KUKA KRL program: EPS_2_251491_MH03A_A_20251118025156.src

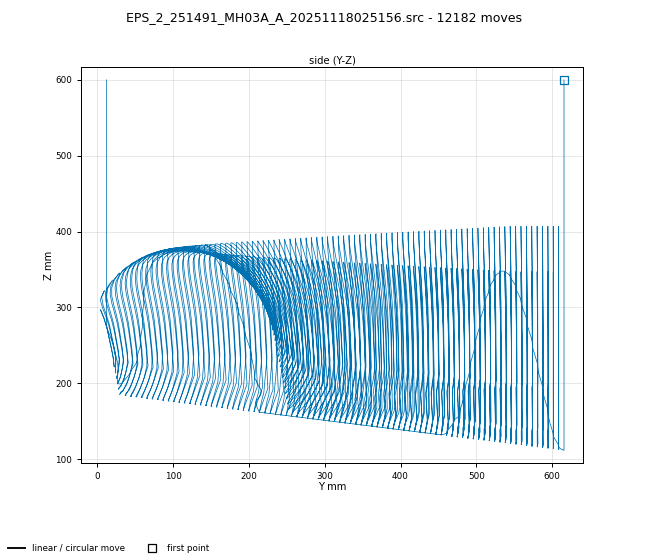
[picture p0: tool path of EPS_2_251491_MH03A_A_20251118025156.src, 12182 of 12184 moves have a stored position in this frame; points joined in program order, loops and branches not executed]
&ACCESS RVP
&REL 4
&COMMENT QRS 19112012
&PARAM EDITMASK = *
DEF PART()
EXT BAS (BAS_COMMAND :IN,REAL :IN )
INT I
BAS (#INITMOV,0 )

;KUKA QRS Post kuka4.cps  Date:22-06-2017 !

File_ID=2917

QRS_PRE_INIT()

;Init var - Until changes are made in qrs_pre_init
Outlet_Square_prg=0
Inlet_1_Square_prg=0
Inlet_2_Square_prg=0
Inlet_3_Square_prg=0
Inlet_4_Square_prg=0
Inlet_5_Square_prg=0

Outlet_1={X 0.000, Y 546.330, Z 306.500, B 0.000, E1 0.000 }
Inlet_1={X 0.000, Y 550.600, Z 246.500, B 0.000, E1 115.000 }
Outlet_1_type=201
Inlet_1_type=201
;QRS#1=Sidecore dimensions
;QRS#2=200-8" PVC SDR 35
;QRS#3=200-8" PVC SDR 35
;QRS#4=
;QRS#5=
;QRS#6=
;QRS#7=
;QRS#8=
;QRS#9=12-08 PSX
;QRS#10=12-08 PSX
;QRS#11=
;QRS#12=
;QRS#13=
;QRS#14=
;QRS#15=
;QRS#16=1220x127x686 2,25'
;QRS#17=EPS Height
;QRS#18=407
;QRS#19=*
;QRS#20= UPDATED VERSION 22-06-2017
;QRS#21=*
Outlet_Square=0100
Inlet_1_Square=0100
Inlet_2_Square=0
Inlet_3_Square=0
Inlet_4_Square=0
Inlet_5_Square=0
Mill_Square=1
Outlet_Square_Prg=204
Inlet_1_Square_prg=204

QRS_INIT()

$ADVANCE=5

; T1
PTP {E1 173.624,E2 173.624}
PTP {X 0,Y 615.49,A -85,B 0,C 180,E1 173.624,E2 173.624,E3 0,E4 0,E5 0,E6 0}
QRS_SPEED_INIT()
LIN {X 0,Y 615.49,Z 600,A -85,B 0,C 180,E1 173.624,E2 173.624,E3 0,E4 0,E5 0,E6 0} C_VEL
LIN {X 0,Y 615.49,Z 121.877,A -85,B 0,C 180,E1 173.624,E2 173.624} C_VEL
LIN {X 0,Y 615.49,Z 113.698,A -85,B 0,C 180,E1 173.624,E2 173.624} C_VEL
LIN {X 0,Y 615.469,Z 111.698,A -85,B 0,C 180,E1 173.438,E2 173.438} C_VEL
LIN {X 0,Y 615.485,Z 111.809,A -85,B 0,C 180,E1 172.29,E2 172.29} C_VEL
LIN {X 0,Y 615.448,Z 127.375,A -85,B 0,C 180,E1 169.473,E2 169.473} C_VEL
LIN {X 0,Y 615.475,Z 136.667,A -85,B 0,C 180,E1 167.805,E2 167.805} C_VEL
LIN {X 0,Y 615.485,Z 242.691,A -85,B 0,C 180,E1 166.547,E2 166.547} C_VEL
LIN {X 0,Y 615.49,Z 256.094,A -85,B 0,C 180,E1 166.252,E2 166.252} C_VEL
LIN {X 0,Y 615.493,Z 268.774,A -85,B 0,C 180,E1 165.836,E2 165.836} C_VEL
LIN {X 0,Y 615.466,Z 281.129,A -85,B 0,C 180,E1 165.282,E2 165.282} C_VEL
LIN {X 0,Y 615.476,Z 292.718,A -85,B 0,C 180,E1 164.604,E2 164.604} C_VEL
LIN {X 0,Y 615.498,Z 303.278,A -85,B 0,C 180,E1 163.831,E2 163.831} C_VEL
LIN {X 0,Y 615.498,Z 311.724,A -85,B 0,C 180,E1 163.072,E2 163.072} C_VEL
LIN {X 0,Y 615.498,Z 321.005,A -85,B 0,C 180,E1 162.044,E2 162.044} C_VEL
LIN {X 0,Y 615.496,Z 328.473,A -85,B 0,C 180,E1 161.009,E2 161.009} C_VEL
LIN {X 0,Y 615.497,Z 334.384,A -85,B 0,C 180,E1 159.968,E2 159.968} C_VEL
LIN {X 0,Y 615.495,Z 339.006,A -85,B 0,C 180,E1 158.92,E2 158.92} C_VEL
LIN {X 0,Y 615.492,Z 343.02,A -85,B 0,C 180,E1 157.653,E2 157.653} C_VEL
LIN {X 0,Y 615.496,Z 345.367,A -85,B 0,C 180,E1 156.444,E2 156.444} C_VEL
LIN {X 0,Y 615.493,Z 346.09,A -85,B 0,C 180,E1 155.729,E2 155.729} C_VEL
LIN {X 0,Y 615.498,Z 346.381,A -85,B 0,C 180,E1 155.009,E2 155.009} C_VEL
LIN {X 0,Y 615.496,Z 346.162,A -85,B 0,C 180,E1 154.285,E2 154.285} C_VEL
LIN {X 0,Y 615.497,Z 344.544,A -85,B 0,C 180,E1 152.954,E2 152.954} C_VEL
LIN {X 0,Y 615.492,Z 342.561,A -85,B 0,C 180,E1 152.085,E2 152.085} C_VEL
LIN {X 0,Y 615.496,Z 338.927,A -85,B 0,C 180,E1 150.969,E2 150.969} C_VEL
LIN {X 0,Y 615.497,Z 333.887,A -85,B 0,C 180,E1 149.841,E2 149.841} C_VEL
LIN {X 0,Y 615.494,Z 328.551,A -85,B 0,C 180,E1 148.913,E2 148.913} C_VEL
LIN {X 0,Y 615.495,Z 320.711,A -85,B 0,C 180,E1 147.83,E2 147.83} C_VEL
LIN {X 0,Y 615.498,Z 312.921,A -85,B 0,C 180,E1 146.96,E2 146.96} C_VEL
LIN {X 0,Y 615.497,Z 303.548,A -85,B 0,C 180,E1 146.101,E2 146.101} C_VEL
LIN {X 0,Y 615.487,Z 292.623,A -85,B 0,C 180,E1 145.3,E2 145.3} C_VEL
LIN {X 0,Y 615.492,Z 282.198,A -85,B 0,C 180,E1 144.686,E2 144.686} C_VEL
LIN {X 0,Y 615.486,Z 271.098,A -85,B 0,C 180,E1 144.167,E2 144.167} C_VEL
LIN {X 0,Y 615.458,Z 258.459,A -85,B 0,C 180,E1 143.722,E2 143.722} C_VEL
LIN {X 0,Y 615.456,Z 245.542,A -85,B 0,C 180,E1 143.415,E2 143.415} C_VEL
LIN {X 0,Y 615.467,Z 226.579,A -85,B 0,C 180,E1 143.161,E2 143.161} C_VEL
LIN {X 0,Y 615.448,Z 136.583,A -85,B 0,C 180,E1 142.089,E2 142.089} C_VEL
LIN {X 0,Y 615.481,Z 123.017,A -85,B 0,C 180,E1 139.654,E2 139.654} C_VEL
LIN {X 0,Y 615.467,Z 111.691,A -85,B 0,C 180,E1 137.559,E2 137.559} C_VEL
LIN {X 0,Y 615.495,Z 111.683,A -85,B 0,C 180,E1 134.933,E2 134.933} C_VEL
LIN {X 0,Y 615.482,Z 111.697,A -85,B 0,C 180,E1 132.08,E2 132.08} C_VEL
LIN {X 0,Y 615.466,Z 111.691,A -85,B 0,C 180,E1 129.752,E2 129.752} C_VEL
LIN {X 0,Y 615.488,Z 111.687,A -85,B 0,C 180,E1 126.937,E2 126.937} C_VEL
LIN {X 0,Y 615.47,Z 111.693,A -85,B 0,C 180,E1 124.023,E2 124.023} C_VEL
LIN {X 0,Y 615.469,Z 111.688,A -85,B 0,C 180,E1 121.687,E2 121.687} C_VEL
LIN {X 0,Y 615.486,Z 111.683,A -85,B 0,C 180,E1 119.407,E2 119.407} C_VEL
LIN {X 0,Y 615.481,Z 111.698,A -85,B 0,C 180,E1 116.445,E2 116.445} C_VEL
LIN {X 0,Y 615.485,Z 111.684,A -85,B 0,C 180,E1 113.557,E2 113.557} C_VEL
LIN {X 0,Y 615.48,Z 111.698,A -85,B 0,C 180,E1 110.556,E2 110.556} C_VEL
LIN {X 0,Y 615.473,Z 111.686,A -85,B 0,C 180,E1 107.958,E2 107.958} C_VEL
LIN {X 0,Y 615.486,Z 111.691,A -85,B 0,C 180,E1 105.226,E2 105.226} C_VEL
LIN {X 0,Y 615.471,Z 111.694,A -85,B 0,C 180,E1 102.531,E2 102.531} C_VEL
LIN {X 0,Y 615.492,Z 111.682,A -85,B 0,C 180,E1 99.862,E2 99.862} C_VEL
LIN {X 0,Y 615.49,Z 111.696,A -85,B 0,C 180,E1 97.216,E2 97.216} C_VEL
LIN {X 0,Y 615.469,Z 111.692,A -85,B 0,C 180,E1 94.585,E2 94.585} C_VEL
LIN {X 0,Y 615.499,Z 111.681,A -85,B 0,C 180,E1 91.963,E2 91.963} C_VEL
LIN {X 0,Y 615.491,Z 111.697,A -85,B 0,C 180,E1 89.346,E2 89.346} C_VEL
LIN {X 0,Y 615.469,Z 111.691,A -85,B 0,C 180,E1 86.727,E2 86.727} C_VEL
LIN {X 0,Y 615.498,Z 111.681,A -85,B 0,C 180,E1 84.102,E2 84.102} C_VEL
LIN {X 0,Y 615.494,Z 111.698,A -85,B 0,C 180,E1 81.464,E2 81.464} C_VEL
LIN {X 0,Y 615.469,Z 111.69,A -85,B 0,C 180,E1 78.807,E2 78.807} C_VEL
LIN {X 0,Y 615.487,Z 111.686,A -85,B 0,C 180,E1 76.066,E2 76.066} C_VEL
LIN {X 0,Y 615.483,Z 111.699,A -85,B 0,C 180,E1 73.414,E2 73.414} C_VEL
LIN {X 0,Y 615.481,Z 111.684,A -85,B 0,C 180,E1 70.662,E2 70.662} C_VEL
LIN {X 0,Y 615.487,Z 111.696,A -85,B 0,C 180,E1 67.864,E2 67.864} C_VEL
LIN {X 0,Y 615.471,Z 111.688,A -85,B 0,C 180,E1 65.008,E2 65.008} C_VEL
LIN {X 0,Y 615.479,Z 111.685,A -85,B 0,C 180,E1 62.823,E2 62.823} C_VEL
LIN {X 0,Y 615.499,Z 111.7,A -85,B 0,C 180,E1 59.841,E2 59.841} C_VEL
LIN {X 0,Y 615.475,Z 111.694,A -85,B 0,C 180,E1 57.542,E2 57.542} C_VEL
LIN {X 0,Y 615.471,Z 111.688,A -85,B 0,C 180,E1 55.184,E2 55.184} C_VEL
LIN {X 0,Y 615.493,Z 111.682,A -85,B 0,C 180,E1 52.759,E2 52.759} C_VEL
LIN {X 0,Y 615.487,Z 111.698,A -85,B 0,C 180,E1 49.911,E2 49.911} C_VEL
LIN {X 0,Y 615.47,Z 111.693,A -85,B 0,C 180,E1 47.646,E2 47.646} C_VEL
LIN {X 0,Y 615.495,Z 111.682,A -85,B 0,C 180,E1 44.933,E2 44.933} C_VEL
LIN {X 0,Y 615.488,Z 111.698,A -85,B 0,C 180,E1 42.081,E2 42.081} C_VEL
LIN {X 0,Y 615.469,Z 111.691,A -85,B 0,C 180,E1 39.751,E2 39.751} C_VEL
LIN {X 0,Y 615.487,Z 111.686,A -85,B 0,C 180,E1 36.937,E2 36.937} C_VEL
LIN {X 0,Y 615.474,Z 111.694,A -85,B 0,C 180,E1 34.022,E2 34.022} C_VEL
LIN {X 0,Y 615.471,Z 111.688,A -85,B 0,C 180,E1 31.686,E2 31.686} C_VEL
LIN {X 0,Y 615.487,Z 111.683,A -85,B 0,C 180,E1 29.406,E2 29.406} C_VEL
LIN {X 0,Y 615.485,Z 111.699,A -85,B 0,C 180,E1 26.444,E2 26.444} C_VEL
LIN {X 0,Y 615.485,Z 111.683,A -85,B 0,C 180,E1 23.556,E2 23.556} C_VEL
LIN {X 0,Y 615.483,Z 111.699,A -85,B 0,C 180,E1 20.557,E2 20.557} C_VEL
LIN {X 0,Y 615.475,Z 111.686,A -85,B 0,C 180,E1 17.957,E2 17.957} C_VEL
LIN {X 0,Y 615.482,Z 111.691,A -85,B 0,C 180,E1 15.226,E2 15.226} C_VEL
LIN {X 0,Y 615.477,Z 111.694,A -85,B 0,C 180,E1 12.53,E2 12.53} C_VEL
LIN {X 0,Y 615.493,Z 111.681,A -85,B 0,C 180,E1 9.862,E2 9.862} C_VEL
LIN {X 0,Y 615.486,Z 111.695,A -85,B 0,C 180,E1 7.215,E2 7.215} C_VEL
LIN {X 0,Y 615.473,Z 111.692,A -85,B 0,C 180,E1 4.584,E2 4.584} C_VEL
LIN {X 0,Y 615.5,Z 111.68,A -85,B 0,C 180,E1 1.963,E2 1.963} C_VEL
LIN {X 0,Y 615.488,Z 111.695,A -85,B 0,C 180,E1 -0.654,E2 -0.654} C_VEL
LIN {X 0,Y 615.473,Z 111.692,A -85,B 0,C 180,E1 -3.273,E2 -3.273} C_VEL
LIN {X 0,Y 615.498,Z 111.681,A -85,B 0,C 180,E1 -5.899,E2 -5.899} C_VEL
LIN {X 0,Y 615.49,Z 111.697,A -85,B 0,C 180,E1 -8.537,E2 -8.537} C_VEL
LIN {X 0,Y 615.472,Z 111.69,A -85,B 0,C 180,E1 -11.194,E2 -11.194} C_VEL
LIN {X 0,Y 615.486,Z 111.686,A -85,B 0,C 180,E1 -13.933,E2 -13.933} C_VEL
LIN {X 0,Y 615.486,Z 111.701,A -85,B 0,C 180,E1 -16.587,E2 -16.587} C_VEL
LIN {X 0,Y 615.482,Z 111.684,A -85,B 0,C 180,E1 -19.338,E2 -19.338} C_VEL
LIN {X 0,Y 615.483,Z 111.695,A -85,B 0,C 180,E1 -22.137,E2 -22.137} C_VEL
LIN {X 0,Y 615.474,Z 111.688,A -85,B 0,C 180,E1 -24.993,E2 -24.993} C_VEL
LIN {X 0,Y 615.481,Z 111.684,A -85,B 0,C 180,E1 -27.178,E2 -27.178} C_VEL
LIN {X 0,Y 615.482,Z 111.69,A -85,B 0,C 180,E1 -29.794,E2 -29.794} C_VEL
LIN {X 0,Y 615.479,Z 111.695,A -85,B 0,C 180,E1 -32.458,E2 -32.458} C_VEL
LIN {X 0,Y 615.475,Z 111.687,A -85,B 0,C 180,E1 -34.816,E2 -34.816} C_VEL
LIN {X 0,Y 615.493,Z 111.682,A -85,B 0,C 180,E1 -37.242,E2 -37.242} C_VEL
LIN {X 0,Y 615.493,Z 111.699,A -85,B 0,C 180,E1 -40.09,E2 -40.09} C_VEL
LIN {X 0,Y 615.488,Z 111.683,A -85,B 0,C 180,E1 -43.048,E2 -43.048} C_VEL
LIN {X 0,Y 615.49,Z 111.698,A -85,B 0,C 180,E1 -46.003,E2 -46.003} C_VEL
LIN {X 0,Y 615.487,Z 111.683,A -85,B 0,C 180,E1 -48.906,E2 -48.906} C_VEL
LIN {X 0,Y 615.485,Z 111.697,A -85,B 0,C 180,E1 -51.932,E2 -51.932} C_VEL
LIN {X 0,Y 615.472,Z 111.688,A -85,B 0,C 180,E1 -54.383,E2 -54.383} C_VEL
LIN {X 0,Y 615.487,Z 111.683,A -85,B 0,C 180,E1 -56.764,E2 -56.764} C_VEL
LIN {X 0,Y 615.482,Z 111.689,A -85,B 0,C 180,E1 -59.08,E2 -59.08} C_VEL
LIN {X 0,Y 615.496,Z 111.701,A -85,B 0,C 180,E1 -61.549,E2 -61.549} C_VEL
LIN {X 0,Y 615.485,Z 111.683,A -85,B 0,C 180,E1 -64.432,E2 -64.432} C_VEL
LIN {X 0,Y 615.488,Z 111.875,A -85,B 0,C 180,E1 -66.711,E2 -66.711} C_VEL
LIN {X 0,Y 615.45,Z 133.105,A -85,B 0,C 180,E1 -69.453,E2 -69.453} C_VEL
LIN {X 0,Y 615.494,Z 154.838,A -85,B 0,C 180,E1 -72.215,E2 -72.215} C_VEL
LIN {X 0,Y 615.485,Z 176.626,A -85,B 0,C 180,E1 -74.944,E2 -74.944} C_VEL
LIN {X 0,Y 615.449,Z 194.138,A -85,B 0,C 180,E1 -77.113,E2 -77.113} C_VEL
LIN {X 0,Y 615.488,Z 302.845,A -85,B 0,C 180,E1 -78.411,E2 -78.411} C_VEL
LIN {X 0,Y 615.477,Z 315.355,A -85,B 0,C 180,E1 -78.682,E2 -78.682} C_VEL
LIN {X 0,Y 615.488,Z 328.618,A -85,B 0,C 180,E1 -79.113,E2 -79.113} C_VEL
LIN {X 0,Y 615.477,Z 340.484,A -85,B 0,C 180,E1 -79.639,E2 -79.639} C_VEL
LIN {X 0,Y 615.494,Z 351.998,A -85,B 0,C 180,E1 -80.304,E2 -80.304} C_VEL
LIN {X 0,Y 615.499,Z 362.344,A -85,B 0,C 180,E1 -81.05,E2 -81.05} C_VEL
LIN {X 0,Y 615.497,Z 370.814,A -85,B 0,C 180,E1 -81.794,E2 -81.794} C_VEL
LIN {X 0,Y 615.498,Z 378.608,A -85,B 0,C 180,E1 -82.62,E2 -82.62} C_VEL
LIN {X 0,Y 615.496,Z 386.205,A -85,B 0,C 180,E1 -83.608,E2 -83.608} C_VEL
LIN {X 0,Y 615.498,Z 393.206,A -85,B 0,C 180,E1 -84.759,E2 -84.759} C_VEL
LIN {X 0,Y 615.494,Z 397.852,A -85,B 0,C 180,E1 -85.744,E2 -85.744} C_VEL
LIN {X 0,Y 615.494,Z 401.399,A -85,B 0,C 180,E1 -86.727,E2 -86.727} C_VEL
LIN {X 0,Y 615.497,Z 403.234,A -85,B 0,C 180,E1 -87.382,E2 -87.382} C_VEL
LIN {X 0,Y 615.5,Z 404.608,A -85,B 0,C 180,E1 -88.037,E2 -88.037} C_VEL
LIN {X 0,Y 615.496,Z 406.174,A -85,B 0,C 180,E1 -89.346,E2 -89.346} C_VEL
LIN {X 0,Y 615.494,Z 406.389,A -85,B 0,C 180,E1 -90,E2 -90} C_VEL
LIN {X 0,Y 615.495,Z 405.58,A -85,B 0,C 180,E1 -91.309,E2 -91.309} C_VEL
LIN {X 0,Y 615.5,Z 404.607,A -85,B 0,C 180,E1 -91.963,E2 -91.963} C_VEL
LIN {X 0,Y 615.497,Z 403.232,A -85,B 0,C 180,E1 -92.618,E2 -92.618} C_VEL
LIN {X 0,Y 615.496,Z 400.349,A -85,B 0,C 180,E1 -93.601,E2 -93.601} C_VEL
LIN {X 0,Y 615.498,Z 396.44,A -85,B 0,C 180,E1 -94.585,E2 -94.585} C_VEL
LIN {X 0,Y 615.499,Z 391.404,A -85,B 0,C 180,E1 -95.57,E2 -95.57} C_VEL
LIN {X 0,Y 615.497,Z 384.87,A -85,B 0,C 180,E1 -96.583,E2 -96.583} C_VEL
LIN {X 0,Y 615.497,Z 377.131,A -85,B 0,C 180,E1 -97.546,E2 -97.546} C_VEL
LIN {X 0,Y 615.498,Z 369.042,A -85,B 0,C 180,E1 -98.371,E2 -98.371} C_VEL
LIN {X 0,Y 615.499,Z 359.164,A -85,B 0,C 180,E1 -99.199,E2 -99.199} C_VEL
LIN {X 0,Y 615.488,Z 347.977,A -85,B 0,C 180,E1 -99.945,E2 -99.945} C_VEL
LIN {X 0,Y 615.482,Z 337.018,A -85,B 0,C 180,E1 -100.527,E2 -100.527} C_VEL
LIN {X 0,Y 615.48,Z 324.487,A -85,B 0,C 180,E1 -101.04,E2 -101.04} C_VEL
LIN {X 0,Y 615.479,Z 312.057,A -85,B 0,C 180,E1 -101.402,E2 -101.402} C_VEL
LIN {X 0,Y 615.493,Z 298.448,A -85,B 0,C 180,E1 -101.652,E2 -101.652} C_VEL
LIN {X 0,Y 615.449,Z 194.134,A -85,B 0,C 180,E1 -102.887,E2 -102.887} C_VEL
LIN {X 0,Y 615.493,Z 171.173,A -85,B 0,C 180,E1 -105.735,E2 -105.735} C_VEL
LIN {X 0,Y 615.469,Z 149.687,A -85,B 0,C 180,E1 -108.436,E2 -108.436} C_VEL
LIN {X 0,Y 615.496,Z 127.565,A -85,B 0,C 180,E1 -111.256,E2 -111.256} C_VEL
LIN {X 0,Y 615.49,Z 111.683,A -85,B 0,C 180,E1 -113.334,E2 -113.334} C_VEL
LIN {X 0,Y 615.481,Z 111.686,A -85,B 0,C 180,E1 -115.716,E2 -115.716} C_VEL
LIN {X 0,Y 615.496,Z 111.699,A -85,B 0,C 180,E1 -118.451,E2 -118.451} C_VEL
LIN {X 0,Y 615.485,Z 111.685,A -85,B 0,C 180,E1 -121.085,E2 -121.085} C_VEL
LIN {X 0,Y 615.483,Z 111.686,A -85,B 0,C 180,E1 -123.533,E2 -123.533} C_VEL
LIN {X 0,Y 615.48,Z 111.695,A -85,B 0,C 180,E1 -126.425,E2 -126.425} C_VEL
LIN {X 0,Y 615.494,Z 111.681,A -85,B 0,C 180,E1 -129.062,E2 -129.062} C_VEL
LIN {X 0,Y 615.488,Z 111.699,A -85,B 0,C 180,E1 -132.08,E2 -132.08} C_VEL
LIN {X 0,Y 615.495,Z 111.682,A -85,B 0,C 180,E1 -135.068,E2 -135.068} C_VEL
LIN {X 0,Y 615.489,Z 111.698,A -85,B 0,C 180,E1 -137.92,E2 -137.92} C_VEL
LIN {X 0,Y 615.469,Z 111.692,A -85,B 0,C 180,E1 -140.248,E2 -140.248} C_VEL
LIN {X 0,Y 615.488,Z 111.687,A -85,B 0,C 180,E1 -143.064,E2 -143.064} C_VEL
LIN {X 0,Y 615.47,Z 111.693,A -85,B 0,C 180,E1 -145.977,E2 -145.977} C_VEL
LIN {X 0,Y 615.468,Z 111.688,A -85,B 0,C 180,E1 -148.313,E2 -148.313} C_VEL
LIN {X 0,Y 615.486,Z 111.684,A -85,B 0,C 180,E1 -150.593,E2 -150.593} C_VEL
LIN {X 0,Y 615.477,Z 111.697,A -85,B 0,C 180,E1 -153.555,E2 -153.555} C_VEL
LIN {X 0,Y 615.464,Z 111.689,A -85,B 0,C 180,E1 -155.997,E2 -155.997} C_VEL
LIN {X 0,Y 615.495,Z 111.685,A -85,B 0,C 180,E1 -158.568,E2 -158.568} C_VEL
LIN {X 0,Y 615.47,Z 111.696,A -85,B 0,C 180,E1 -161.401,E2 -161.401} C_VEL
LIN {X 0,Y 615.475,Z 111.686,A -85,B 0,C 180,E1 -164.094,E2 -164.094} C_VEL
LIN {X 0,Y 615.493,Z 111.698,A -85,B 0,C 180,E1 -166.799,E2 -166.799} C_VEL
LIN {X 0,Y 615.455,Z 111.693,A -85,B 0,C 180,E1 -169.472,E2 -169.472} C_VEL
LIN {X 0,Y 615.484,Z 111.687,A -85,B 0,C 180,E1 -172.124,E2 -172.124} C_VEL
LIN {X 0,Y 615.488,Z 111.699,A -85,B 0,C 180,E1 -174.759,E2 -174.759} C_VEL
LIN {X 0,Y 615.452,Z 111.692,A -85,B 0,C 180,E1 -177.382,E2 -177.382} C_VEL
LIN {X 0,Y 615.487,Z 111.688,A -85,B 0,C 180,E1 -180,E2 -180} C_VEL
LIN {X 0,Y 615.477,Z 111.698,A -85,B 0,C 180,E1 -182.618,E2 -182.618} C_VEL
LIN {X 0,Y 615.447,Z 111.692,A -85,B 0,C 180,E1 -185.241,E2 -185.241} C_VEL
LIN {X 0,Y 615.469,Z 111.698,A -85,B 0,C 180,E1 -186.562,E2 -186.562} C_VEL
LIN {X 0,Y 614.782,Z 111.892,A -85,B 0,C 180,E1 -186.929,E2 -186.929} C_VEL
LIN {X 0,Y 611.98,Z 112.983,A -85,B 0,C 180,E1 -187.496,E2 -187.496} C_VEL
LIN {X 0,Y 609.163,Z 115.021,A -85,B 0,C 180,E1 -188.047,E2 -188.047} C_VEL
LIN {X 0,Y 608.467,Z 116.714,A -85,B 0,C 180,E1 -188.385,E2 -188.385} C_VEL
LIN {X 0,Y 608.47,Z 131.376,A -85,B 0,C 180,E1 -191.052,E2 -191.052} C_VEL
LIN {X 0,Y 608.452,Z 136.863,A -85,B 0,C 180,E1 -192.042,E2 -192.042} C_VEL
LIN {X 0,Y 608.548,Z 243.573,A -85,B 0,C 180,E1 -193.333,E2 -193.333} C_VEL
LIN {X 0,Y 608.539,Z 256.703,A -85,B 0,C 180,E1 -193.631,E2 -193.631} C_VEL
LIN {X 0,Y 608.522,Z 268.854,A -85,B 0,C 180,E1 -194.036,E2 -194.036} C_VEL
LIN {X 0,Y 608.487,Z 280.346,A -85,B 0,C 180,E1 -194.549,E2 -194.549} C_VEL
LIN {X 0,Y 608.457,Z 292.172,A -85,B 0,C 180,E1 -195.234,E2 -195.234} C_VEL
LIN {X 0,Y 608.477,Z 302.792,A -85,B 0,C 180,E1 -196.007,E2 -196.007} C_VEL
LIN {X 0,Y 608.461,Z 311.53,A -85,B 0,C 180,E1 -196.784,E2 -196.784} C_VEL
LIN {X 0,Y 608.458,Z 320.967,A -85,B 0,C 180,E1 -197.823,E2 -197.823} C_VEL
LIN {X 0,Y 608.447,Z 328.574,A -85,B 0,C 180,E1 -198.87,E2 -198.87} C_VEL
LIN {X 0,Y 608.436,Z 334.624,A -85,B 0,C 180,E1 -199.922,E2 -199.922} C_VEL
LIN {X 0,Y 608.426,Z 339.347,A -85,B 0,C 180,E1 -200.982,E2 -200.982} C_VEL
LIN {X 0,Y 608.454,Z 342.881,A -85,B 0,C 180,E1 -202.048,E2 -202.048} C_VEL
LIN {X 0,Y 608.423,Z 345.311,A -85,B 0,C 180,E1 -203.125,E2 -203.125} C_VEL
LIN {X 0,Y 608.42,Z 346.613,A -85,B 0,C 180,E1 -204.14,E2 -204.14} C_VEL
LIN {X 0,Y 608.439,Z 346.946,A -85,B 0,C 180,E1 -205.301,E2 -205.301} C_VEL
LIN {X 0,Y 608.425,Z 346.552,A -85,B 0,C 180,E1 -206.036,E2 -206.036} C_VEL
LIN {X 0,Y 608.437,Z 344.89,A -85,B 0,C 180,E1 -207.199,E2 -207.199} C_VEL
LIN {X 0,Y 608.427,Z 341.138,A -85,B 0,C 180,E1 -208.612,E2 -208.612} C_VEL
LIN {X 0,Y 608.446,Z 336.505,A -85,B 0,C 180,E1 -209.78,E2 -209.78} C_VEL
LIN {X 0,Y 608.454,Z 330.52,A -85,B 0,C 180,E1 -210.904,E2 -210.904} C_VEL
LIN {X 0,Y 608.466,Z 323.827,A -85,B 0,C 180,E1 -211.899,E2 -211.899} C_VEL
LIN {X 0,Y 608.479,Z 315.688,A -85,B 0,C 180,E1 -212.878,E2 -212.878} C_VEL
LIN {X 0,Y 608.489,Z 306.888,A -85,B 0,C 180,E1 -213.737,E2 -213.737} C_VEL
LIN {X 0,Y 608.477,Z 296.262,A -85,B 0,C 180,E1 -214.578,E2 -214.578} C_VEL
LIN {X 0,Y 608.494,Z 285.309,A -85,B 0,C 180,E1 -215.274,E2 -215.274} C_VEL
LIN {X 0,Y 608.515,Z 273,A -85,B 0,C 180,E1 -215.883,E2 -215.883} C_VEL
LIN {X 0,Y 608.502,Z 260.618,A -85,B 0,C 180,E1 -216.344,E2 -216.344} C_VEL
LIN {X 0,Y 608.501,Z 247.794,A -85,B 0,C 180,E1 -216.679,E2 -216.679} C_VEL
LIN {X 0,Y 608.53,Z 232.344,A -85,B 0,C 180,E1 -216.909,E2 -216.909} C_VEL
LIN {X 0,Y 608.416,Z 136.878,A -85,B 0,C 180,E1 -218.046,E2 -218.046} C_VEL
LIN {X 0,Y 608.482,Z 123.216,A -85,B 0,C 180,E1 -220.517,E2 -220.517} C_VEL
LIN {X 0,Y 608.449,Z 112.69,A -85,B 0,C 180,E1 -222.445,E2 -222.445} C_VEL
LIN {X 0,Y 608.462,Z 112.688,A -85,B 0,C 180,E1 -225.204,E2 -225.204} C_VEL
LIN {X 0,Y 608.462,Z 112.693,A -85,B 0,C 180,E1 -227.938,E2 -227.938} C_VEL
LIN {X 0,Y 608.448,Z 112.688,A -85,B 0,C 180,E1 -230.705,E2 -230.705} C_VEL
LIN {X 0,Y 608.459,Z 112.689,A -85,B 0,C 180,E1 -233.085,E2 -233.085} C_VEL
LIN {X 0,Y 608.466,Z 112.696,A -85,B 0,C 180,E1 -235.53,E2 -235.53} C_VEL
LIN {X 0,Y 608.461,Z 112.69,A -85,B 0,C 180,E1 -237.905,E2 -237.905} C_VEL
LIN {X 0,Y 608.455,Z 112.688,A -85,B 0,C 180,E1 -240.22,E2 -240.22} C_VEL
LIN {X 0,Y 608.48,Z 112.686,A -85,B 0,C 180,E1 -242.792,E2 -242.792} C_VEL
LIN {X 0,Y 608.447,Z 112.697,A -85,B 0,C 180,E1 -245.428,E2 -245.428} C_VEL
LIN {X 0,Y 608.467,Z 112.686,A -85,B 0,C 180,E1 -248.308,E2 -248.308} C_VEL
LIN {X 0,Y 608.468,Z 112.695,A -85,B 0,C 180,E1 -251.284,E2 -251.284} C_VEL
LIN {X 0,Y 608.451,Z 112.688,A -85,B 0,C 180,E1 -253.906,E2 -253.906} C_VEL
LIN {X 0,Y 608.464,Z 112.689,A -85,B 0,C 180,E1 -256.643,E2 -256.643} C_VEL
LIN {X 0,Y 608.455,Z 112.692,A -85,B 0,C 180,E1 -259.35,E2 -259.35} C_VEL
LIN {X 0,Y 608.475,Z 112.685,A -85,B 0,C 180,E1 -262.033,E2 -262.033} C_VEL
LIN {X 0,Y 608.468,Z 112.692,A -85,B 0,C 180,E1 -264.698,E2 -264.698} C_VEL
LIN {X 0,Y 608.463,Z 112.689,A -85,B 0,C 180,E1 -267.352,E2 -267.352} C_VEL
LIN {X 0,Y 608.477,Z 112.685,A -85,B 0,C 180,E1 -270,E2 -270} C_VEL
LIN {X 0,Y 608.478,Z 112.693,A -85,B 0,C 180,E1 -272.648,E2 -272.648} C_VEL
LIN {X 0,Y 608.451,Z 112.689,A -85,B 0,C 180,E1 -275.302,E2 -275.302} C_VEL
LIN {X 0,Y 608.479,Z 112.685,A -85,B 0,C 180,E1 -277.967,E2 -277.967} C_VEL
LIN {X 0,Y 608.463,Z 112.69,A -85,B 0,C 180,E1 -280.954,E2 -280.954} C_VEL
LIN {X 0,Y 608.453,Z 112.688,A -85,B 0,C 180,E1 -283.356,E2 -283.356} C_VEL
LIN {X 0,Y 608.462,Z 112.691,A -85,B 0,C 180,E1 -286.093,E2 -286.093} C_VEL
LIN {X 0,Y 608.452,Z 112.691,A -85,B 0,C 180,E1 -288.869,E2 -288.869} C_VEL
LIN {X 0,Y 608.472,Z 112.686,A -85,B 0,C 180,E1 -291.691,E2 -291.691} C_VEL
LIN {X 0,Y 608.448,Z 112.694,A -85,B 0,C 180,E1 -294.571,E2 -294.571} C_VEL
LIN {X 0,Y 608.472,Z 112.685,A -85,B 0,C 180,E1 -297.207,E2 -297.207} C_VEL
LIN {X 0,Y 608.47,Z 112.692,A -85,B 0,C 180,E1 -299.972,E2 -299.972} C_VEL
LIN {X 0,Y 608.452,Z 112.691,A -85,B 0,C 180,E1 -302.521,E2 -302.521} C_VEL
LIN {X 0,Y 608.438,Z 112.689,A -85,B 0,C 180,E1 -304.904,E2 -304.904} C_VEL
LIN {X 0,Y 608.479,Z 112.684,A -85,B 0,C 180,E1 -307.16,E2 -307.16} C_VEL
LIN {X 0,Y 608.476,Z 112.687,A -85,B 0,C 180,E1 -309.439,E2 -309.439} C_VEL
LIN {X 0,Y 608.442,Z 112.692,A -85,B 0,C 180,E1 -312.333,E2 -312.333} C_VEL
LIN {X 0,Y 608.459,Z 112.687,A -85,B 0,C 180,E1 -314.795,E2 -314.795} C_VEL
LIN {X 0,Y 608.462,Z 112.695,A -85,B 0,C 180,E1 -317.665,E2 -317.665} C_VEL
LIN {X 0,Y 608.475,Z 112.685,A -85,B 0,C 180,E1 -320.701,E2 -320.701} C_VEL
LIN {X 0,Y 608.458,Z 112.689,A -85,B 0,C 180,E1 -323.086,E2 -323.086} C_VEL
LIN {X 0,Y 608.466,Z 112.695,A -85,B 0,C 180,E1 -325.531,E2 -325.531} C_VEL
LIN {X 0,Y 608.465,Z 112.691,A -85,B 0,C 180,E1 -327.906,E2 -327.906} C_VEL
LIN {X 0,Y 608.455,Z 112.688,A -85,B 0,C 180,E1 -330.22,E2 -330.22} C_VEL
LIN {X 0,Y 608.478,Z 112.685,A -85,B 0,C 180,E1 -332.792,E2 -332.792} C_VEL
LIN {X 0,Y 608.447,Z 112.699,A -85,B 0,C 180,E1 -335.429,E2 -335.429} C_VEL
LIN {X 0,Y 608.468,Z 112.686,A -85,B 0,C 180,E1 -338.309,E2 -338.309} C_VEL
LIN {X 0,Y 608.469,Z 112.696,A -85,B 0,C 180,E1 -341.283,E2 -341.283} C_VEL
LIN {X 0,Y 608.453,Z 112.688,A -85,B 0,C 180,E1 -343.906,E2 -343.906} C_VEL
LIN {X 0,Y 608.462,Z 112.689,A -85,B 0,C 180,E1 -346.644,E2 -346.644} C_VEL
LIN {X 0,Y 608.458,Z 112.693,A -85,B 0,C 180,E1 -349.35,E2 -349.35} C_VEL
LIN {X 0,Y 608.476,Z 112.685,A -85,B 0,C 180,E1 -352.033,E2 -352.033} C_VEL
LIN {X 0,Y 608.464,Z 112.692,A -85,B 0,C 180,E1 -354.698,E2 -354.698} C_VEL
LIN {X 0,Y 608.466,Z 112.69,A -85,B 0,C 180,E1 -357.352,E2 -357.352} C_VEL
LIN {X 0,Y 608.477,Z 112.685,A -85,B 0,C 180,E1 -360,E2 -360} C_VEL
LIN {X 0,Y 608.473,Z 112.692,A -85,B 0,C 180,E1 -362.648,E2 -362.648} C_VEL
LIN {X 0,Y 608.454,Z 112.69,A -85,B 0,C 180,E1 -365.302,E2 -365.302} C_VEL
LIN {X 0,Y 608.479,Z 112.685,A -85,B 0,C 180,E1 -367.967,E2 -367.967} C_VEL
LIN {X 0,Y 608.466,Z 112.691,A -85,B 0,C 180,E1 -370.956,E2 -370.956} C_VEL
LIN {X 0,Y 608.455,Z 112.688,A -85,B 0,C 180,E1 -373.357,E2 -373.357} C_VEL
LIN {X 0,Y 608.461,Z 112.69,A -85,B 0,C 180,E1 -376.094,E2 -376.094} C_VEL
LIN {X 0,Y 608.455,Z 112.691,A -85,B 0,C 180,E1 -378.87,E2 -378.87} C_VEL
LIN {X 0,Y 608.471,Z 112.686,A -85,B 0,C 180,E1 -381.692,E2 -381.692} C_VEL
LIN {X 0,Y 608.45,Z 112.694,A -85,B 0,C 180,E1 -384.571,E2 -384.571} C_VEL
LIN {X 0,Y 608.474,Z 112.685,A -85,B 0,C 180,E1 -387.207,E2 -387.207} C_VEL
LIN {X 0,Y 608.468,Z 112.692,A -85,B 0,C 180,E1 -389.972,E2 -389.972} C_VEL
LIN {X 0,Y 608.455,Z 112.688,A -85,B 0,C 180,E1 -392.88,E2 -392.88} C_VEL
LIN {X 0,Y 608.435,Z 112.69,A -85,B 0,C 180,E1 -395.278,E2 -395.278} C_VEL
LIN {X 0,Y 608.471,Z 112.69,A -85,B 0,C 180,E1 -397.746,E2 -397.746} C_VEL
LIN {X 0,Y 608.449,Z 112.693,A -85,B 0,C 180,E1 -400.329,E2 -400.329} C_VEL
LIN {X 0,Y 608.453,Z 112.687,A -85,B 0,C 180,E1 -402.96,E2 -402.96} C_VEL
LIN {X 0,Y 608.465,Z 112.694,A -85,B 0,C 180,E1 -405.736,E2 -405.736} C_VEL
LIN {X 0,Y 608.457,Z 112.687,A -85,B 0,C 180,E1 -408.659,E2 -408.659} C_VEL
LIN {X 0,Y 608.469,Z 112.69,A -85,B 0,C 180,E1 -411.412,E2 -411.412} C_VEL
LIN {X 0,Y 608.445,Z 112.695,A -85,B 0,C 180,E1 -413.955,E2 -413.955} C_VEL
LIN {X 0,Y 608.447,Z 112.689,A -85,B 0,C 180,E1 -416.329,E2 -416.329} C_VEL
LIN {X 0,Y 608.448,Z 112.688,A -85,B 0,C 180,E1 -418.733,E2 -418.733} C_VEL
LIN {X 0,Y 608.476,Z 112.692,A -85,B 0,C 180,E1 -421.38,E2 -421.38} C_VEL
LIN {X 0,Y 608.443,Z 112.692,A -85,B 0,C 180,E1 -423.965,E2 -423.965} C_VEL
LIN {X 0,Y 608.467,Z 112.728,A -85,B 0,C 180,E1 -426.539,E2 -426.539} C_VEL
LIN {X 0,Y 608.595,Z 127.57,A -85,B 0,C 180,E1 -428.491,E2 -428.491} C_VEL
LIN {X 0,Y 608.498,Z 149.174,A -85,B 0,C 180,E1 -431.277,E2 -431.277} C_VEL
LIN {X 0,Y 608.495,Z 168.58,A -85,B 0,C 180,E1 -433.744,E2 -433.744} C_VEL
LIN {X 0,Y 608.479,Z 190.348,A -85,B 0,C 180,E1 -436.474,E2 -436.474} C_VEL
LIN {X 0,Y 608.446,Z 194.357,A -85,B 0,C 180,E1 -436.973,E2 -436.973} C_VEL
LIN {X 0,Y 608.546,Z 302.961,A -85,B 0,C 180,E1 -438.277,E2 -438.277} C_VEL
LIN {X 0,Y 608.512,Z 316.226,A -85,B 0,C 180,E1 -438.572,E2 -438.572} C_VEL
LIN {X 0,Y 608.514,Z 328.631,A -85,B 0,C 180,E1 -438.982,E2 -438.982} C_VEL
LIN {X 0,Y 608.499,Z 340.64,A -85,B 0,C 180,E1 -439.519,E2 -439.519} C_VEL
LIN {X 0,Y 608.484,Z 352.201,A -85,B 0,C 180,E1 -440.191,E2 -440.191} C_VEL
LIN {X 0,Y 608.485,Z 362.597,A -85,B 0,C 180,E1 -440.946,E2 -440.946} C_VEL
LIN {X 0,Y 608.475,Z 371.114,A -85,B 0,C 180,E1 -441.699,E2 -441.699} C_VEL
LIN {X 0,Y 608.471,Z 378.962,A -85,B 0,C 180,E1 -442.534,E2 -442.534} C_VEL
LIN {X 0,Y 608.46,Z 386.288,A -85,B 0,C 180,E1 -443.485,E2 -443.485} C_VEL
LIN {X 0,Y 608.451,Z 391.867,A -85,B 0,C 180,E1 -444.366,E2 -444.366} C_VEL
LIN {X 0,Y 608.432,Z 396.951,A -85,B 0,C 180,E1 -445.362,E2 -445.362} C_VEL
LIN {X 0,Y 608.449,Z 400.897,A -85,B 0,C 180,E1 -446.358,E2 -446.358} C_VEL
LIN {X 0,Y 608.425,Z 403.81,A -85,B 0,C 180,E1 -447.352,E2 -447.352} C_VEL
LIN {X 0,Y 608.445,Z 405.202,A -85,B 0,C 180,E1 -448.014,E2 -448.014} C_VEL
LIN {X 0,Y 608.438,Z 406.784,A -85,B 0,C 180,E1 -449.338,E2 -449.338} C_VEL
LIN {X 0,Y 608.434,Z 407,A -85,B 0,C 180,E1 -450,E2 -450} C_VEL
LIN {X 0,Y 608.448,Z 406.184,A -85,B 0,C 180,E1 -451.324,E2 -451.324} C_VEL
LIN {X 0,Y 608.445,Z 405.201,A -85,B 0,C 180,E1 -451.986,E2 -451.986} C_VEL
LIN {X 0,Y 608.425,Z 403.809,A -85,B 0,C 180,E1 -452.649,E2 -452.649} C_VEL
LIN {X 0,Y 608.449,Z 400.895,A -85,B 0,C 180,E1 -453.643,E2 -453.643} C_VEL
LIN {X 0,Y 608.432,Z 396.949,A -85,B 0,C 180,E1 -454.638,E2 -454.638} C_VEL
LIN {X 0,Y 608.438,Z 390.875,A -85,B 0,C 180,E1 -455.801,E2 -455.801} C_VEL
LIN {X 0,Y 608.462,Z 384.233,A -85,B 0,C 180,E1 -456.8,E2 -456.8} C_VEL
LIN {X 0,Y 608.456,Z 375.987,A -85,B 0,C 180,E1 -457.8,E2 -457.8} C_VEL
LIN {X 0,Y 608.472,Z 367.534,A -85,B 0,C 180,E1 -458.636,E2 -458.636} C_VEL
LIN {X 0,Y 608.479,Z 357.088,A -85,B 0,C 180,E1 -459.474,E2 -459.474} C_VEL
LIN {X 0,Y 608.489,Z 346.752,A -85,B 0,C 180,E1 -460.145,E2 -460.145} C_VEL
LIN {X 0,Y 608.519,Z 335.263,A -85,B 0,C 180,E1 -460.74,E2 -460.74} C_VEL
LIN {X 0,Y 608.528,Z 322.885,A -85,B 0,C 180,E1 -461.225,E2 -461.225} C_VEL
LIN {X 0,Y 608.544,Z 309.428,A -85,B 0,C 180,E1 -461.597,E2 -461.597} C_VEL
LIN {X 0,Y 608.553,Z 297.066,A -85,B 0,C 180,E1 -461.808,E2 -461.808} C_VEL
LIN {X 0,Y 608.434,Z 194.268,A -85,B 0,C 180,E1 -463.039,E2 -463.039} C_VEL
LIN {X 0,Y 608.523,Z 171.237,A -85,B 0,C 180,E1 -465.92,E2 -465.92} C_VEL
LIN {X 0,Y 608.53,Z 150.969,A -85,B 0,C 180,E1 -468.492,E2 -468.492} C_VEL
LIN {X 0,Y 608.571,Z 130.295,A -85,B 0,C 180,E1 -471.155,E2 -471.155} C_VEL
LIN {X 0,Y 608.521,Z 112.894,A -85,B 0,C 180,E1 -473.437,E2 -473.437} C_VEL
LIN {X 0,Y 608.472,Z 112.691,A -85,B 0,C 180,E1 -474.151,E2 -474.151} C_VEL
LIN {X 0,Y 608.448,Z 112.693,A -85,B 0,C 180,E1 -476.775,E2 -476.775} C_VEL
LIN {X 0,Y 608.471,Z 112.687,A -85,B 0,C 180,E1 -479.02,E2 -479.02} C_VEL
LIN {X 0,Y 608.448,Z 112.688,A -85,B 0,C 180,E1 -481.318,E2 -481.318} C_VEL
LIN {X 0,Y 608.476,Z 112.688,A -85,B 0,C 180,E1 -483.735,E2 -483.735} C_VEL
LIN {X 0,Y 608.447,Z 112.698,A -85,B 0,C 180,E1 -486.092,E2 -486.092} C_VEL
LIN {X 0,Y 608.469,Z 112.688,A -85,B 0,C 180,E1 -488.588,E2 -488.588} C_VEL
LIN {X 0,Y 608.461,Z 112.688,A -85,B 0,C 180,E1 -491.342,E2 -491.342} C_VEL
LIN {X 0,Y 608.453,Z 112.692,A -85,B 0,C 180,E1 -494.263,E2 -494.263} C_VEL
LIN {X 0,Y 608.455,Z 112.688,A -85,B 0,C 180,E1 -497.04,E2 -497.04} C_VEL
LIN {X 0,Y 608.456,Z 112.697,A -85,B 0,C 180,E1 -499.697,E2 -499.697} C_VEL
LIN {X 0,Y 608.465,Z 112.688,A -85,B 0,C 180,E1 -502.253,E2 -502.253} C_VEL
LIN {X 0,Y 608.449,Z 112.691,A -85,B 0,C 180,E1 -505.095,E2 -505.095} C_VEL
LIN {X 0,Y 608.46,Z 112.69,A -85,B 0,C 180,E1 -507.905,E2 -507.905} C_VEL
LIN {X 0,Y 608.454,Z 112.688,A -85,B 0,C 180,E1 -510.219,E2 -510.219} C_VEL
LIN {X 0,Y 608.482,Z 112.686,A -85,B 0,C 180,E1 -512.792,E2 -512.792} C_VEL
LIN {X 0,Y 608.445,Z 112.696,A -85,B 0,C 180,E1 -515.428,E2 -515.428} C_VEL
LIN {X 0,Y 608.466,Z 112.686,A -85,B 0,C 180,E1 -518.308,E2 -518.308} C_VEL
LIN {X 0,Y 608.464,Z 112.693,A -85,B 0,C 180,E1 -521.287,E2 -521.287} C_VEL
LIN {X 0,Y 608.445,Z 112.689,A -85,B 0,C 180,E1 -523.906,E2 -523.906} C_VEL
LIN {X 0,Y 608.467,Z 112.692,A -85,B 0,C 180,E1 -526.643,E2 -526.643} C_VEL
LIN {X 0,Y 608.44,Z 112.692,A -85,B 0,C 180,E1 -529.349,E2 -529.349} C_VEL
LIN {X 0,Y 608.473,Z 112.686,A -85,B 0,C 180,E1 -532.033,E2 -532.033} C_VEL
LIN {X 0,Y 608.468,Z 112.696,A -85,B 0,C 180,E1 -534.698,E2 -534.698} C_VEL
LIN {X 0,Y 608.447,Z 112.689,A -85,B 0,C 180,E1 -537.352,E2 -537.352} C_VEL
LIN {X 0,Y 608.477,Z 112.687,A -85,B 0,C 180,E1 -540,E2 -540} C_VEL
LIN {X 0,Y 608.467,Z 112.692,A -85,B 0,C 180,E1 -542.648,E2 -542.648} C_VEL
LIN {X 0,Y 608.433,Z 112.69,A -85,B 0,C 180,E1 -545.302,E2 -545.302} C_VEL
LIN {X 0,Y 608.472,Z 112.84,A -85,B 0,C 180,E1 -547.675,E2 -547.675} C_VEL
LIN {X 0,Y 608.467,Z 116.714,A -85,B 0,C 180,E1 -548.385,E2 -548.385} C_VEL
LIN {X 0,Y 607.75,Z 119.486,A -85,B 0,C 180,E1 -548.872,E2 -548.872} C_VEL
LIN {X 0,Y 602.018,Z 128.867,A -85,B 0,C 180,E1 -550.44,E2 -550.44} C_VEL
LIN {X 0,Y 601.405,Z 131.649,A -85,B 0,C 180,E1 -550.935,E2 -550.935} C_VEL
LIN {X 0,Y 601.42,Z 136.85,A -85,B 0,C 180,E1 -551.885,E2 -551.885} C_VEL
LIN {X 0,Y 601.677,Z 144.218,A -85,B 0,C 180,E1 -551.988,E2 -551.988} C_VEL
LIN {X 0,Y 601.603,Z 243.211,A -85,B 0,C 180,E1 -553.189,E2 -553.189} C_VEL
LIN {X 0,Y 601.59,Z 256.429,A -85,B 0,C 180,E1 -553.49,E2 -553.49} C_VEL
LIN {X 0,Y 601.555,Z 269.229,A -85,B 0,C 180,E1 -553.921,E2 -553.921} C_VEL
LIN {X 0,Y 601.501,Z 281.031,A -85,B 0,C 180,E1 -554.462,E2 -554.462} C_VEL
LIN {X 0,Y 601.428,Z 292.735,A -85,B 0,C 180,E1 -555.157,E2 -555.157} C_VEL
LIN {X 0,Y 601.437,Z 303.253,A -85,B 0,C 180,E1 -555.938,E2 -555.938} C_VEL
LIN {X 0,Y 601.409,Z 312.228,A -85,B 0,C 180,E1 -556.756,E2 -556.756} C_VEL
LIN {X 0,Y 601.385,Z 320.571,A -85,B 0,C 180,E1 -557.688,E2 -557.688} C_VEL
LIN {X 0,Y 601.374,Z 327.276,A -85,B 0,C 180,E1 -558.601,E2 -558.601} C_VEL
LIN {X 0,Y 601.383,Z 332.46,A -85,B 0,C 180,E1 -559.454,E2 -559.454} C_VEL
LIN {X 0,Y 601.354,Z 337.671,A -85,B 0,C 180,E1 -560.524,E2 -560.524} C_VEL
LIN {X 0,Y 601.343,Z 341.65,A -85,B 0,C 180,E1 -561.601,E2 -561.601} C_VEL
LIN {X 0,Y 601.32,Z 344.505,A -85,B 0,C 180,E1 -562.686,E2 -562.686} C_VEL
LIN {X 0,Y 601.32,Z 345.818,A -85,B 0,C 180,E1 -563.414,E2 -563.414} C_VEL
LIN {X 0,Y 601.321,Z 346.71,A -85,B 0,C 180,E1 -564.268,E2 -564.268} C_VEL
LIN {X 0,Y 601.337,Z 346.968,A -85,B 0,C 180,E1 -564.881,E2 -564.881} C_VEL
LIN {X 0,Y 601.335,Z 346.689,A -85,B 0,C 180,E1 -565.852,E2 -565.852} C_VEL
LIN {X 0,Y 601.334,Z 345.1,A -85,B 0,C 180,E1 -567.117,E2 -567.117} C_VEL
LIN {X 0,Y 601.341,Z 342.401,A -85,B 0,C 180,E1 -568.251,E2 -568.251} C_VEL
LIN {X 0,Y 601.352,Z 338.387,A -85,B 0,C 180,E1 -569.396,E2 -569.396} C_VEL
LIN {X 0,Y 601.365,Z 332.894,A -85,B 0,C 180,E1 -570.555,E2 -570.555} C_VEL
LIN {X 0,Y 601.395,Z 325.678,A -85,B 0,C 180,E1 -571.727,E2 -571.727} C_VEL
LIN {X 0,Y 601.402,Z 317.17,A -85,B 0,C 180,E1 -572.802,E2 -572.802} C_VEL
LIN {X 0,Y 601.437,Z 308.259,A -85,B 0,C 180,E1 -573.714,E2 -573.714} C_VEL
LIN {X 0,Y 601.449,Z 298.578,A -85,B 0,C 180,E1 -574.522,E2 -574.522} C_VEL
LIN {X 0,Y 601.487,Z 286.626,A -85,B 0,C 180,E1 -575.317,E2 -575.317} C_VEL
LIN {X 0,Y 601.514,Z 274.914,A -85,B 0,C 180,E1 -575.925,E2 -575.925} C_VEL
LIN {X 0,Y 601.537,Z 262.314,A -85,B 0,C 180,E1 -576.421,E2 -576.421} C_VEL
LIN {X 0,Y 601.549,Z 248.797,A -85,B 0,C 180,E1 -576.794,E2 -576.794} C_VEL
LIN {X 0,Y 601.58,Z 235.211,A -85,B 0,C 180,E1 -577.014,E2 -577.014} C_VEL
LIN {X 0,Y 601.533,Z 138.058,A -85,B 0,C 180,E1 -578.179,E2 -578.179} C_VEL
LIN {X 0,Y 601.383,Z 136.825,A -85,B 0,C 180,E1 -578.21,E2 -578.21} C_VEL
LIN {X 0,Y 601.449,Z 122.304,A -85,B 0,C 180,E1 -580.871,E2 -580.871} C_VEL
LIN {X 0,Y 601.429,Z 113.565,A -85,B 0,C 180,E1 -582.498,E2 -582.498} C_VEL
LIN {X 0,Y 601.426,Z 113.569,A -85,B 0,C 180,E1 -585.482,E2 -585.482} C_VEL
LIN {X 0,Y 601.42,Z 113.564,A -85,B 0,C 180,E1 -588.407,E2 -588.407} C_VEL
LIN {X 0,Y 601.43,Z 113.571,A -85,B 0,C 180,E1 -591.529,E2 -591.529} C_VEL
LIN {X 0,Y 601.382,Z 113.569,A -85,B 0,C 180,E1 -594.245,E2 -594.245} C_VEL
LIN {X 0,Y 601.417,Z 113.564,A -85,B 0,C 180,E1 -596.686,E2 -596.686} C_VEL
LIN {X 0,Y 601.412,Z 113.568,A -85,B 0,C 180,E1 -599.057,E2 -599.057} C_VEL
LIN {X 0,Y 601.431,Z 113.572,A -85,B 0,C 180,E1 -601.373,E2 -601.373} C_VEL
LIN {X 0,Y 601.398,Z 113.572,A -85,B 0,C 180,E1 -603.636,E2 -603.636} C_VEL
LIN {X 0,Y 601.417,Z 113.565,A -85,B 0,C 180,E1 -606.589,E2 -606.589} C_VEL
LIN {X 0,Y 601.426,Z 113.569,A -85,B 0,C 180,E1 -609.478,E2 -609.478} C_VEL
LIN {X 0,Y 601.392,Z 113.567,A -85,B 0,C 180,E1 -612.311,E2 -612.311} C_VEL
LIN {X 0,Y 601.411,Z 113.565,A -85,B 0,C 180,E1 -614.408,E2 -614.408} C_VEL
LIN {X 0,Y 601.413,Z 113.574,A -85,B 0,C 180,E1 -617.171,E2 -617.171} C_VEL
LIN {X 0,Y 601.433,Z 113.562,A -85,B 0,C 180,E1 -619.905,E2 -619.905} C_VEL
LIN {X 0,Y 601.442,Z 113.565,A -85,B 0,C 180,E1 -622.615,E2 -622.615} C_VEL
LIN {X 0,Y 601.41,Z 113.569,A -85,B 0,C 180,E1 -625.308,E2 -625.308} C_VEL
LIN {X 0,Y 601.437,Z 113.562,A -85,B 0,C 180,E1 -627.991,E2 -627.991} C_VEL
LIN {X 0,Y 601.455,Z 113.567,A -85,B 0,C 180,E1 -630.669,E2 -630.669} C_VEL
LIN {X 0,Y 601.417,Z 113.566,A -85,B 0,C 180,E1 -633.349,E2 -633.349} C_VEL
LIN {X 0,Y 601.442,Z 113.562,A -85,B 0,C 180,E1 -636.037,E2 -636.037} C_VEL
LIN {X 0,Y 601.437,Z 113.57,A -85,B 0,C 180,E1 -638.737,E2 -638.737} C_VEL
LIN {X 0,Y 601.411,Z 113.565,A -85,B 0,C 180,E1 -641.458,E2 -641.458} C_VEL
LIN {X 0,Y 601.418,Z 113.569,A -85,B 0,C 180,E1 -644.205,E2 -644.205} C_VEL
LIN {X 0,Y 601.428,Z 113.565,A -85,B 0,C 180,E1 -646.986,E2 -646.986} C_VEL
LIN {X 0,Y 601.403,Z 113.568,A -85,B 0,C 180,E1 -649.809,E2 -649.809} C_VEL
LIN {X 0,Y 601.409,Z 113.569,A -85,B 0,C 180,E1 -652.683,E2 -652.683} C_VEL
LIN {X 0,Y 601.398,Z 113.568,A -85,B 0,C 180,E1 -654.878,E2 -654.878} C_VEL
LIN {X 0,Y 601.412,Z 113.565,A -85,B 0,C 180,E1 -657.362,E2 -657.362} C_VEL
LIN {X 0,Y 601.447,Z 113.571,A -85,B 0,C 180,E1 -660.163,E2 -660.163} C_VEL
LIN {X 0,Y 601.415,Z 113.566,A -85,B 0,C 180,E1 -662.715,E2 -662.715} C_VEL
LIN {X 0,Y 601.388,Z 113.567,A -85,B 0,C 180,E1 -665.111,E2 -665.111} C_VEL
LIN {X 0,Y 601.434,Z 113.564,A -85,B 0,C 180,E1 -667.419,E2 -667.419} C_VEL
LIN {X 0,Y 601.409,Z 113.575,A -85,B 0,C 180,E1 -669.995,E2 -669.995} C_VEL
LIN {X 0,Y 601.407,Z 113.566,A -85,B 0,C 180,E1 -672.67,E2 -672.67} C_VEL
LIN {X 0,Y 601.423,Z 113.568,A -85,B 0,C 180,E1 -675.482,E2 -675.482} C_VEL
LIN {X 0,Y 601.421,Z 113.565,A -85,B 0,C 180,E1 -678.407,E2 -678.407} C_VEL
LIN {X 0,Y 601.435,Z 113.562,A -85,B 0,C 180,E1 -680.876,E2 -680.876} C_VEL
LIN {X 0,Y 601.402,Z 113.572,A -85,B 0,C 180,E1 -683.417,E2 -683.417} C_VEL
LIN {X 0,Y 601.429,Z 113.566,A -85,B 0,C 180,E1 -686.064,E2 -686.064} C_VEL
LIN {X 0,Y 601.438,Z 113.561,A -85,B 0,C 180,E1 -688.542,E2 -688.542} C_VEL
LIN {X 0,Y 601.433,Z 113.57,A -85,B 0,C 180,E1 -691.374,E2 -691.374} C_VEL
LIN {X 0,Y 601.4,Z 113.573,A -85,B 0,C 180,E1 -693.636,E2 -693.636} C_VEL
LIN {X 0,Y 601.416,Z 113.564,A -85,B 0,C 180,E1 -696.59,E2 -696.59} C_VEL
LIN {X 0,Y 601.427,Z 113.57,A -85,B 0,C 180,E1 -699.478,E2 -699.478} C_VEL
LIN {X 0,Y 601.392,Z 113.567,A -85,B 0,C 180,E1 -702.312,E2 -702.312} C_VEL
LIN {X 0,Y 601.41,Z 113.565,A -85,B 0,C 180,E1 -704.409,E2 -704.409} C_VEL
LIN {X 0,Y 601.415,Z 113.575,A -85,B 0,C 180,E1 -707.172,E2 -707.172} C_VEL
LIN {X 0,Y 601.435,Z 113.562,A -85,B 0,C 180,E1 -709.905,E2 -709.905} C_VEL
LIN {X 0,Y 601.44,Z 113.565,A -85,B 0,C 180,E1 -712.615,E2 -712.615} C_VEL
LIN {X 0,Y 601.412,Z 113.569,A -85,B 0,C 180,E1 -715.308,E2 -715.308} C_VEL
LIN {X 0,Y 601.437,Z 113.561,A -85,B 0,C 180,E1 -717.991,E2 -717.991} C_VEL
LIN {X 0,Y 601.452,Z 113.567,A -85,B 0,C 180,E1 -720.67,E2 -720.67} C_VEL
LIN {X 0,Y 601.42,Z 113.566,A -85,B 0,C 180,E1 -723.35,E2 -723.35} C_VEL
LIN {X 0,Y 601.442,Z 113.562,A -85,B 0,C 180,E1 -726.037,E2 -726.037} C_VEL
LIN {X 0,Y 601.436,Z 113.571,A -85,B 0,C 180,E1 -728.738,E2 -728.738} C_VEL
LIN {X 0,Y 601.421,Z 113.564,A -85,B 0,C 180,E1 -731.459,E2 -731.459} C_VEL
LIN {X 0,Y 601.419,Z 113.568,A -85,B 0,C 180,E1 -734.206,E2 -734.206} C_VEL
LIN {X 0,Y 601.429,Z 113.565,A -85,B 0,C 180,E1 -736.986,E2 -736.986} C_VEL
LIN {X 0,Y 601.403,Z 113.567,A -85,B 0,C 180,E1 -739.81,E2 -739.81} C_VEL
LIN {X 0,Y 601.414,Z 113.571,A -85,B 0,C 180,E1 -742.606,E2 -742.606} C_VEL
LIN {X 0,Y 601.4,Z 113.568,A -85,B 0,C 180,E1 -744.879,E2 -744.879} C_VEL
LIN {X 0,Y 601.413,Z 113.564,A -85,B 0,C 180,E1 -747.363,E2 -747.363} C_VEL
LIN {X 0,Y 601.428,Z 113.572,A -85,B 0,C 180,E1 -750.164,E2 -750.164} C_VEL
LIN {X 0,Y 601.419,Z 113.566,A -85,B 0,C 180,E1 -752.715,E2 -752.715} C_VEL
LIN {X 0,Y 601.39,Z 113.567,A -85,B 0,C 180,E1 -755.112,E2 -755.112} C_VEL
LIN {X 0,Y 601.436,Z 113.563,A -85,B 0,C 180,E1 -757.419,E2 -757.419} C_VEL
LIN {X 0,Y 601.411,Z 113.575,A -85,B 0,C 180,E1 -759.995,E2 -759.995} C_VEL
LIN {X 0,Y 601.41,Z 113.566,A -85,B 0,C 180,E1 -762.671,E2 -762.671} C_VEL
LIN {X 0,Y 601.427,Z 113.566,A -85,B 0,C 180,E1 -765.482,E2 -765.482} C_VEL
LIN {X 0,Y 601.424,Z 113.565,A -85,B 0,C 180,E1 -768.407,E2 -768.407} C_VEL
LIN {X 0,Y 601.437,Z 113.562,A -85,B 0,C 180,E1 -770.876,E2 -770.876} C_VEL
LIN {X 0,Y 601.404,Z 113.571,A -85,B 0,C 180,E1 -773.417,E2 -773.417} C_VEL
LIN {X 0,Y 601.432,Z 113.566,A -85,B 0,C 180,E1 -776.065,E2 -776.065} C_VEL
LIN {X 0,Y 601.42,Z 113.564,A -85,B 0,C 180,E1 -778.546,E2 -778.546} C_VEL
LIN {X 0,Y 601.436,Z 113.569,A -85,B 0,C 180,E1 -781.374,E2 -781.374} C_VEL
LIN {X 0,Y 601.402,Z 113.575,A -85,B 0,C 180,E1 -783.637,E2 -783.637} C_VEL
LIN {X 0,Y 601.428,Z 113.581,A -85,B 0,C 180,E1 -786.362,E2 -786.362} C_VEL
LIN {X 0,Y 601.75,Z 116.652,A -85,B 0,C 180,E1 -786.786,E2 -786.786} C_VEL
LIN {X 0,Y 601.612,Z 138.488,A -85,B 0,C 180,E1 -789.663,E2 -789.663} C_VEL
LIN {X 0,Y 601.549,Z 160.323,A -85,B 0,C 180,E1 -792.492,E2 -792.492} C_VEL
LIN {X 0,Y 601.46,Z 180.795,A -85,B 0,C 180,E1 -795.104,E2 -795.104} C_VEL
LIN {X 0,Y 601.42,Z 194.357,A -85,B 0,C 180,E1 -796.818,E2 -796.818} C_VEL
LIN {X 0,Y 601.629,Z 207.686,A -85,B 0,C 180,E1 -796.984,E2 -796.984} C_VEL
LIN {X 0,Y 601.613,Z 302.961,A -85,B 0,C 180,E1 -798.14,E2 -798.14} C_VEL
LIN {X 0,Y 601.56,Z 316.227,A -85,B 0,C 180,E1 -798.438,E2 -798.438} C_VEL
LIN {X 0,Y 601.545,Z 327.908,A -85,B 0,C 180,E1 -798.825,E2 -798.825} C_VEL
LIN {X 0,Y 601.522,Z 340.638,A -85,B 0,C 180,E1 -799.396,E2 -799.396} C_VEL
LIN {X 0,Y 601.483,Z 352.203,A -85,B 0,C 180,E1 -800.076,E2 -800.076} C_VEL
LIN {X 0,Y 601.444,Z 362.599,A -85,B 0,C 180,E1 -800.839,E2 -800.839} C_VEL
LIN {X 0,Y 601.429,Z 371.115,A -85,B 0,C 180,E1 -801.601,E2 -801.601} C_VEL
LIN {X 0,Y 601.418,Z 378.963,A -85,B 0,C 180,E1 -802.446,E2 -802.446} C_VEL
LIN {X 0,Y 601.37,Z 386.226,A -85,B 0,C 180,E1 -803.398,E2 -803.398} C_VEL
LIN {X 0,Y 601.372,Z 391.868,A -85,B 0,C 180,E1 -804.299,E2 -804.299} C_VEL
LIN {X 0,Y 601.336,Z 396.951,A -85,B 0,C 180,E1 -805.308,E2 -805.308} C_VEL
LIN {X 0,Y 601.368,Z 400.897,A -85,B 0,C 180,E1 -806.315,E2 -806.315} C_VEL
LIN {X 0,Y 601.325,Z 403.81,A -85,B 0,C 180,E1 -807.321,E2 -807.321} C_VEL
LIN {X 0,Y 601.343,Z 405.202,A -85,B 0,C 180,E1 -807.991,E2 -807.991} C_VEL
LIN {X 0,Y 601.339,Z 406.784,A -85,B 0,C 180,E1 -809.331,E2 -809.331} C_VEL
LIN {X 0,Y 601.335,Z 407,A -85,B 0,C 180,E1 -810,E2 -810} C_VEL
LIN {X 0,Y 601.347,Z 406.184,A -85,B 0,C 180,E1 -811.34,E2 -811.34} C_VEL
LIN {X 0,Y 601.343,Z 405.202,A -85,B 0,C 180,E1 -812.01,E2 -812.01} C_VEL
LIN {X 0,Y 601.325,Z 403.809,A -85,B 0,C 180,E1 -812.68,E2 -812.68} C_VEL
LIN {X 0,Y 601.368,Z 400.895,A -85,B 0,C 180,E1 -813.686,E2 -813.686} C_VEL
LIN {X 0,Y 601.336,Z 396.949,A -85,B 0,C 180,E1 -814.693,E2 -814.693} C_VEL
LIN {X 0,Y 601.373,Z 390.876,A -85,B 0,C 180,E1 -815.869,E2 -815.869} C_VEL
LIN {X 0,Y 601.382,Z 384.234,A -85,B 0,C 180,E1 -816.88,E2 -816.88} C_VEL
LIN {X 0,Y 601.4,Z 375.987,A -85,B 0,C 180,E1 -817.893,E2 -817.893} C_VEL
LIN {X 0,Y 601.436,Z 367.534,A -85,B 0,C 180,E1 -818.738,E2 -818.738} C_VEL
LIN {X 0,Y 601.449,Z 357.09,A -85,B 0,C 180,E1 -819.585,E2 -819.585} C_VEL
LIN {X 0,Y 601.467,Z 346.754,A -85,B 0,C 180,E1 -820.265,E2 -820.265} C_VEL
LIN {X 0,Y 601.538,Z 334.597,A -85,B 0,C 180,E1 -820.896,E2 -820.896} C_VEL
LIN {X 0,Y 601.555,Z 322.211,A -85,B 0,C 180,E1 -821.379,E2 -821.379} C_VEL
LIN {X 0,Y 601.583,Z 309.427,A -85,B 0,C 180,E1 -821.733,E2 -821.733} C_VEL
LIN {X 0,Y 601.623,Z 297.066,A -85,B 0,C 180,E1 -821.946,E2 -821.946} C_VEL
LIN {X 0,Y 601.531,Z 195.123,A -85,B 0,C 180,E1 -823.17,E2 -823.17} C_VEL
LIN {X 0,Y 601.426,Z 194.268,A -85,B 0,C 180,E1 -823.193,E2 -823.193} C_VEL
LIN {X 0,Y 601.512,Z 171.237,A -85,B 0,C 180,E1 -826.111,E2 -826.111} C_VEL
LIN {X 0,Y 601.575,Z 151.697,A -85,B 0,C 180,E1 -828.62,E2 -828.62} C_VEL
LIN {X 0,Y 601.667,Z 130.295,A -85,B 0,C 180,E1 -831.409,E2 -831.409} C_VEL
LIN {X 0,Y 601.724,Z 115.283,A -85,B 0,C 180,E1 -833.398,E2 -833.398} C_VEL
LIN {X 0,Y 601.422,Z 113.568,A -85,B 0,C 180,E1 -833.661,E2 -833.661} C_VEL
LIN {X 0,Y 601.403,Z 113.575,A -85,B 0,C 180,E1 -836.364,E2 -836.364} C_VEL
LIN {X 0,Y 601.441,Z 113.566,A -85,B 0,C 180,E1 -838.789,E2 -838.789} C_VEL
LIN {X 0,Y 601.423,Z 113.564,A -85,B 0,C 180,E1 -841.455,E2 -841.455} C_VEL
LIN {X 0,Y 601.429,Z 113.571,A -85,B 0,C 180,E1 -844.119,E2 -844.119} C_VEL
LIN {X 0,Y 601.44,Z 113.562,A -85,B 0,C 180,E1 -847.382,E2 -847.382} C_VEL
LIN {X 0,Y 601.406,Z 113.576,A -85,B 0,C 180,E1 -849.996,E2 -849.996} C_VEL
LIN {X 0,Y 601.412,Z 113.566,A -85,B 0,C 180,E1 -852.671,E2 -852.671} C_VEL
LIN {X 0,Y 601.43,Z 113.567,A -85,B 0,C 180,E1 -855.482,E2 -855.482} C_VEL
LIN {X 0,Y 601.424,Z 113.565,A -85,B 0,C 180,E1 -858.407,E2 -858.407} C_VEL
LIN {X 0,Y 601.433,Z 113.57,A -85,B 0,C 180,E1 -861.529,E2 -861.529} C_VEL
LIN {X 0,Y 601.384,Z 113.569,A -85,B 0,C 180,E1 -864.245,E2 -864.245} C_VEL
LIN {X 0,Y 601.419,Z 113.564,A -85,B 0,C 180,E1 -866.686,E2 -866.686} C_VEL
LIN {X 0,Y 601.414,Z 113.568,A -85,B 0,C 180,E1 -869.057,E2 -869.057} C_VEL
LIN {X 0,Y 601.432,Z 113.573,A -85,B 0,C 180,E1 -871.373,E2 -871.373} C_VEL
LIN {X 0,Y 601.398,Z 113.571,A -85,B 0,C 180,E1 -873.636,E2 -873.636} C_VEL
LIN {X 0,Y 601.441,Z 113.563,A -85,B 0,C 180,E1 -875.859,E2 -875.859} C_VEL
LIN {X 0,Y 601.409,Z 113.569,A -85,B 0,C 180,E1 -878.761,E2 -878.761} C_VEL
LIN {X 0,Y 601.394,Z 113.569,A -85,B 0,C 180,E1 -881.607,E2 -881.607} C_VEL
LIN {X 0,Y 601.412,Z 113.567,A -85,B 0,C 180,E1 -884.408,E2 -884.408} C_VEL
LIN {X 0,Y 601.408,Z 113.571,A -85,B 0,C 180,E1 -887.171,E2 -887.171} C_VEL
LIN {X 0,Y 601.428,Z 113.563,A -85,B 0,C 180,E1 -889.905,E2 -889.905} C_VEL
LIN {X 0,Y 601.441,Z 113.57,A -85,B 0,C 180,E1 -892.615,E2 -892.615} C_VEL
LIN {X 0,Y 601.397,Z 113.568,A -85,B 0,C 180,E1 -895.308,E2 -895.308} C_VEL
LIN {X 0,Y 601.436,Z 113.564,A -85,B 0,C 180,E1 -897.991,E2 -897.991} C_VEL
LIN {X 0,Y 601.442,Z 113.568,A -85,B 0,C 180,E1 -900.669,E2 -900.669} C_VEL
LIN {X 0,Y 601.376,Z 113.57,A -85,B 0,C 180,E1 -903.35,E2 -903.35} C_VEL
LIN {X 0,Y 601.437,Z 113.568,A -85,B 0,C 180,E1 -906.037,E2 -906.037} C_VEL
LIN {X 0,Y 601.45,Z 113.769,A -85,B 0,C 180,E1 -907.638,E2 -907.638} C_VEL
LIN {X 0,Y 601.403,Z 128.925,A -85,B 0,C 180,E1 -910.436,E2 -910.436} C_VEL
LIN {X 0,Y 601.405,Z 131.649,A -85,B 0,C 180,E1 -910.935,E2 -910.935} C_VEL
LIN {X 0,Y 601.124,Z 133.892,A -85,B 0,C 180,E1 -911.227,E2 -911.227} C_VEL
LIN {X 0,Y 600.132,Z 137.598,A -85,B 0,C 180,E1 -911.507,E2 -911.507} C_VEL
LIN {X 0,Y 598.765,Z 141.866,A -85,B 0,C 180,E1 -911.703,E2 -911.703} C_VEL
LIN {X 0,Y 596.958,Z 147.56,A -85,B 0,C 180,E1 -911.854,E2 -911.854} C_VEL
LIN {X 0,Y 595.078,Z 155.647,A -85,B 0,C 180,E1 -911.974,E2 -911.974} C_VEL
LIN {X 0,Y 594.737,Z 159.793,A -85,B 0,C 180,E1 -912.022,E2 -912.022} C_VEL
LIN {X 0,Y 594.652,Z 242.845,A -85,B 0,C 180,E1 -913.042,E2 -913.042} C_VEL
LIN {X 0,Y 594.628,Z 255.398,A -85,B 0,C 180,E1 -913.325,E2 -913.325} C_VEL
LIN {X 0,Y 594.561,Z 267.846,A -85,B 0,C 180,E1 -913.736,E2 -913.736} C_VEL
LIN {X 0,Y 594.507,Z 280.307,A -85,B 0,C 180,E1 -914.297,E2 -914.297} C_VEL
LIN {X 0,Y 594.453,Z 291.961,A -85,B 0,C 180,E1 -914.988,E2 -914.988} C_VEL
LIN {X 0,Y 594.396,Z 301.542,A -85,B 0,C 180,E1 -915.692,E2 -915.692} C_VEL
LIN {X 0,Y 594.365,Z 310.474,A -85,B 0,C 180,E1 -916.486,E2 -916.486} C_VEL
LIN {X 0,Y 594.35,Z 318.702,A -85,B 0,C 180,E1 -917.372,E2 -917.372} C_VEL
LIN {X 0,Y 594.315,Z 326.731,A -85,B 0,C 180,E1 -918.441,E2 -918.441} C_VEL
LIN {X 0,Y 594.296,Z 332.187,A -85,B 0,C 180,E1 -919.337,E2 -919.337} C_VEL
LIN {X 0,Y 594.283,Z 337.447,A -85,B 0,C 180,E1 -920.418,E2 -920.418} C_VEL
LIN {X 0,Y 594.249,Z 341.479,A -85,B 0,C 180,E1 -921.507,E2 -921.507} C_VEL
LIN {X 0,Y 594.243,Z 344.602,A -85,B 0,C 180,E1 -922.707,E2 -922.707} C_VEL
LIN {X 0,Y 594.22,Z 346.205,A -85,B 0,C 180,E1 -923.711,E2 -923.711} C_VEL
LIN {X 0,Y 594.241,Z 346.828,A -85,B 0,C 180,E1 -924.452,E2 -924.452} C_VEL
LIN {X 0,Y 594.224,Z 346.971,A -85,B 0,C 180,E1 -925.2,E2 -925.2} C_VEL
LIN {X 0,Y 594.227,Z 346.601,A -85,B 0,C 180,E1 -925.991,E2 -925.991} C_VEL
LIN {X 0,Y 594.226,Z 345.793,A -85,B 0,C 180,E1 -926.707,E2 -926.707} C_VEL
LIN {X 0,Y 594.269,Z 344.346,A -85,B 0,C 180,E1 -927.504,E2 -927.504} C_VEL
LIN {X 0,Y 594.246,Z 341.474,A -85,B 0,C 180,E1 -928.584,E2 -928.584} C_VEL
LIN {X 0,Y 594.277,Z 336.991,A -85,B 0,C 180,E1 -929.781,E2 -929.781} C_VEL
LIN {X 0,Y 594.28,Z 331.028,A -85,B 0,C 180,E1 -930.959,E2 -930.959} C_VEL
LIN {X 0,Y 594.343,Z 324.244,A -85,B 0,C 180,E1 -932.005,E2 -932.005} C_VEL
LIN {X 0,Y 594.349,Z 316.668,A -85,B 0,C 180,E1 -932.952,E2 -932.952} C_VEL
LIN {X 0,Y 594.378,Z 308.84,A -85,B 0,C 180,E1 -933.761,E2 -933.761} C_VEL
LIN {X 0,Y 594.427,Z 299.333,A -85,B 0,C 180,E1 -934.577,E2 -934.577} C_VEL
LIN {X 0,Y 594.485,Z 287.292,A -85,B 0,C 180,E1 -935.399,E2 -935.399} C_VEL
LIN {X 0,Y 594.53,Z 275.596,A -85,B 0,C 180,E1 -936.022,E2 -936.022} C_VEL
LIN {X 0,Y 594.566,Z 263.761,A -85,B 0,C 180,E1 -936.506,E2 -936.506} C_VEL
LIN {X 0,Y 594.625,Z 250.501,A -85,B 0,C 180,E1 -936.893,E2 -936.893} C_VEL
LIN {X 0,Y 594.653,Z 237.487,A -85,B 0,C 180,E1 -937.127,E2 -937.127} C_VEL
LIN {X 0,Y 594.66,Z 138.932,A -85,B 0,C 180,E1 -938.323,E2 -938.323} C_VEL
LIN {X 0,Y 594.315,Z 136.783,A -85,B 0,C 180,E1 -938.378,E2 -938.378} C_VEL
LIN {X 0,Y 594.418,Z 122.037,A -85,B 0,C 180,E1 -941.113,E2 -941.113} C_VEL
LIN {X 0,Y 594.397,Z 114.441,A -85,B 0,C 180,E1 -942.551,E2 -942.551} C_VEL
LIN {X 0,Y 594.364,Z 114.445,A -85,B 0,C 180,E1 -945.191,E2 -945.191} C_VEL
LIN {X 0,Y 594.381,Z 114.444,A -85,B 0,C 180,E1 -948.152,E2 -948.152} C_VEL
LIN {X 0,Y 594.379,Z 114.444,A -85,B 0,C 180,E1 -951.194,E2 -951.194} C_VEL
LIN {X 0,Y 594.35,Z 114.452,A -85,B 0,C 180,E1 -953.755,E2 -953.755} C_VEL
LIN {X 0,Y 594.364,Z 114.443,A -85,B 0,C 180,E1 -956.238,E2 -956.238} C_VEL
LIN {X 0,Y 594.369,Z 114.442,A -85,B 0,C 180,E1 -958.649,E2 -958.649} C_VEL
LIN {X 0,Y 594.383,Z 114.444,A -85,B 0,C 180,E1 -961.042,E2 -961.042} C_VEL
LIN {X 0,Y 594.381,Z 114.442,A -85,B 0,C 180,E1 -963.978,E2 -963.978} C_VEL
LIN {X 0,Y 594.384,Z 114.44,A -85,B 0,C 180,E1 -966.295,E2 -966.295} C_VEL
LIN {X 0,Y 594.403,Z 114.448,A -85,B 0,C 180,E1 -969.224,E2 -969.224} C_VEL
LIN {X 0,Y 594.344,Z 114.445,A -85,B 0,C 180,E1 -972.094,E2 -972.094} C_VEL
LIN {X 0,Y 594.362,Z 114.443,A -85,B 0,C 180,E1 -974.219,E2 -974.219} C_VEL
LIN {X 0,Y 594.382,Z 114.441,A -85,B 0,C 180,E1 -976.321,E2 -976.321} C_VEL
LIN {X 0,Y 594.372,Z 114.451,A -85,B 0,C 180,E1 -979.094,E2 -979.094} C_VEL
LIN {X 0,Y 594.41,Z 114.437,A -85,B 0,C 180,E1 -981.843,E2 -981.843} C_VEL
LIN {X 0,Y 594.4,Z 114.443,A -85,B 0,C 180,E1 -984.572,E2 -984.572} C_VEL
LIN {X 0,Y 594.398,Z 114.442,A -85,B 0,C 180,E1 -987.289,E2 -987.289} C_VEL
LIN {X 0,Y 594.414,Z 114.437,A -85,B 0,C 180,E1 -990,E2 -990} C_VEL
LIN {X 0,Y 594.408,Z 114.447,A -85,B 0,C 180,E1 -992.711,E2 -992.711} C_VEL
LIN {X 0,Y 594.388,Z 114.44,A -85,B 0,C 180,E1 -995.428,E2 -995.428} C_VEL
LIN {X 0,Y 594.418,Z 114.439,A -85,B 0,C 180,E1 -998.156,E2 -998.156} C_VEL
LIN {X 0,Y 594.388,Z 114.442,A -85,B 0,C 180,E1 -1001.074,E2 -1001.074} C_VEL
LIN {X 0,Y 594.377,Z 114.441,A -85,B 0,C 180,E1 -1003.679,E2 -1003.679} C_VEL
LIN {X 0,Y 594.394,Z 114.445,A -85,B 0,C 180,E1 -1006.72,E2 -1006.72} C_VEL
LIN {X 0,Y 594.365,Z 114.442,A -85,B 0,C 180,E1 -1009.334,E2 -1009.334} C_VEL
LIN {X 0,Y 594.367,Z 114.442,A -85,B 0,C 180,E1 -1011.503,E2 -1011.503} C_VEL
LIN {X 0,Y 594.387,Z 114.447,A -85,B 0,C 180,E1 -1014.446,E2 -1014.446} C_VEL
LIN {X 0,Y 594.38,Z 114.444,A -85,B 0,C 180,E1 -1016.699,E2 -1016.699} C_VEL
LIN {X 0,Y 594.378,Z 114.441,A -85,B 0,C 180,E1 -1018.998,E2 -1018.998} C_VEL
LIN {X 0,Y 594.389,Z 114.442,A -85,B 0,C 180,E1 -1021.645,E2 -1021.645} C_VEL
LIN {X 0,Y 594.374,Z 114.444,A -85,B 0,C 180,E1 -1024.58,E2 -1024.58} C_VEL
LIN {X 0,Y 594.384,Z 114.44,A -85,B 0,C 180,E1 -1027.086,E2 -1027.086} C_VEL
LIN {X 0,Y 594.374,Z 114.448,A -85,B 0,C 180,E1 -1029.775,E2 -1029.775} C_VEL
LIN {X 0,Y 594.364,Z 114.446,A -85,B 0,C 180,E1 -1032.375,E2 -1032.375} C_VEL
LIN {X 0,Y 594.36,Z 114.444,A -85,B 0,C 180,E1 -1035.191,E2 -1035.191} C_VEL
LIN {X 0,Y 594.381,Z 114.445,A -85,B 0,C 180,E1 -1038.151,E2 -1038.151} C_VEL
LIN {X 0,Y 594.385,Z 114.442,A -85,B 0,C 180,E1 -1041.195,E2 -1041.195} C_VEL
LIN {X 0,Y 594.349,Z 114.453,A -85,B 0,C 180,E1 -1043.756,E2 -1043.756} C_VEL
LIN {X 0,Y 594.374,Z 114.443,A -85,B 0,C 180,E1 -1046.239,E2 -1046.239} C_VEL
LIN {X 0,Y 594.387,Z 114.44,A -85,B 0,C 180,E1 -1048.651,E2 -1048.651} C_VEL
LIN {X 0,Y 594.381,Z 114.444,A -85,B 0,C 180,E1 -1051.042,E2 -1051.042} C_VEL
LIN {X 0,Y 594.382,Z 114.443,A -85,B 0,C 180,E1 -1053.977,E2 -1053.977} C_VEL
LIN {X 0,Y 594.384,Z 114.44,A -85,B 0,C 180,E1 -1056.296,E2 -1056.296} C_VEL
LIN {X 0,Y 594.403,Z 114.446,A -85,B 0,C 180,E1 -1059.225,E2 -1059.225} C_VEL
LIN {X 0,Y 594.349,Z 114.445,A -85,B 0,C 180,E1 -1062.095,E2 -1062.095} C_VEL
LIN {X 0,Y 594.362,Z 114.443,A -85,B 0,C 180,E1 -1064.219,E2 -1064.219} C_VEL
LIN {X 0,Y 594.38,Z 114.441,A -85,B 0,C 180,E1 -1066.321,E2 -1066.321} C_VEL
LIN {X 0,Y 594.374,Z 114.452,A -85,B 0,C 180,E1 -1069.095,E2 -1069.095} C_VEL
LIN {X 0,Y 594.41,Z 114.437,A -85,B 0,C 180,E1 -1071.844,E2 -1071.844} C_VEL
LIN {X 0,Y 594.396,Z 114.442,A -85,B 0,C 180,E1 -1074.573,E2 -1074.573} C_VEL
LIN {X 0,Y 594.4,Z 114.443,A -85,B 0,C 180,E1 -1077.289,E2 -1077.289} C_VEL
LIN {X 0,Y 594.414,Z 114.436,A -85,B 0,C 180,E1 -1080,E2 -1080} C_VEL
LIN {X 0,Y 594.404,Z 114.446,A -85,B 0,C 180,E1 -1082.711,E2 -1082.711} C_VEL
LIN {X 0,Y 594.39,Z 114.44,A -85,B 0,C 180,E1 -1085.428,E2 -1085.428} C_VEL
LIN {X 0,Y 594.417,Z 114.438,A -85,B 0,C 180,E1 -1088.157,E2 -1088.157} C_VEL
LIN {X 0,Y 594.389,Z 114.443,A -85,B 0,C 180,E1 -1091.075,E2 -1091.075} C_VEL
LIN {X 0,Y 594.378,Z 114.441,A -85,B 0,C 180,E1 -1093.679,E2 -1093.679} C_VEL
LIN {X 0,Y 594.394,Z 114.446,A -85,B 0,C 180,E1 -1096.72,E2 -1096.72} C_VEL
LIN {X 0,Y 594.366,Z 114.442,A -85,B 0,C 180,E1 -1099.335,E2 -1099.335} C_VEL
LIN {X 0,Y 594.367,Z 114.442,A -85,B 0,C 180,E1 -1101.504,E2 -1101.504} C_VEL
LIN {X 0,Y 594.388,Z 114.448,A -85,B 0,C 180,E1 -1104.446,E2 -1104.446} C_VEL
LIN {X 0,Y 594.382,Z 114.444,A -85,B 0,C 180,E1 -1106.7,E2 -1106.7} C_VEL
LIN {X 0,Y 594.38,Z 114.441,A -85,B 0,C 180,E1 -1108.999,E2 -1108.999} C_VEL
LIN {X 0,Y 594.377,Z 114.443,A -85,B 0,C 180,E1 -1111.643,E2 -1111.643} C_VEL
LIN {X 0,Y 594.376,Z 114.444,A -85,B 0,C 180,E1 -1114.58,E2 -1114.58} C_VEL
LIN {X 0,Y 594.391,Z 114.442,A -85,B 0,C 180,E1 -1117.609,E2 -1117.609} C_VEL
LIN {X 0,Y 594.37,Z 114.444,A -85,B 0,C 180,E1 -1120.567,E2 -1120.567} C_VEL
LIN {X 0,Y 594.367,Z 114.444,A -85,B 0,C 180,E1 -1123.3,E2 -1123.3} C_VEL
LIN {X 0,Y 594.369,Z 114.447,A -85,B 0,C 180,E1 -1126.161,E2 -1126.161} C_VEL
LIN {X 0,Y 594.381,Z 114.441,A -85,B 0,C 180,E1 -1128.537,E2 -1128.537} C_VEL
LIN {X 0,Y 594.388,Z 114.442,A -85,B 0,C 180,E1 -1131.296,E2 -1131.296} C_VEL
LIN {X 0,Y 594.352,Z 114.454,A -85,B 0,C 180,E1 -1133.756,E2 -1133.756} C_VEL
LIN {X 0,Y 594.377,Z 114.443,A -85,B 0,C 180,E1 -1136.239,E2 -1136.239} C_VEL
LIN {X 0,Y 594.37,Z 114.442,A -85,B 0,C 180,E1 -1138.65,E2 -1138.65} C_VEL
LIN {X 0,Y 594.385,Z 114.443,A -85,B 0,C 180,E1 -1141.042,E2 -1141.042} C_VEL
LIN {X 0,Y 594.385,Z 114.444,A -85,B 0,C 180,E1 -1143.978,E2 -1143.978} C_VEL
LIN {X 0,Y 594.396,Z 114.525,A -85,B 0,C 180,E1 -1146.204,E2 -1146.204} C_VEL
LIN {X 0,Y 594.863,Z 118.016,A -85,B 0,C 180,E1 -1146.685,E2 -1146.685} C_VEL
LIN {X 0,Y 594.693,Z 139.852,A -85,B 0,C 180,E1 -1149.597,E2 -1149.597} C_VEL
LIN {X 0,Y 594.579,Z 163.053,A -85,B 0,C 180,E1 -1152.635,E2 -1152.635} C_VEL
LIN {X 0,Y 594.465,Z 183.524,A -85,B 0,C 180,E1 -1155.275,E2 -1155.275} C_VEL
LIN {X 0,Y 594.422,Z 194.357,A -85,B 0,C 180,E1 -1156.66,E2 -1156.66} C_VEL
LIN {X 0,Y 594.749,Z 200.531,A -85,B 0,C 180,E1 -1156.743,E2 -1156.743} C_VEL
LIN {X 0,Y 594.665,Z 302.961,A -85,B 0,C 180,E1 -1157.999,E2 -1157.999} C_VEL
LIN {X 0,Y 594.601,Z 316.228,A -85,B 0,C 180,E1 -1158.301,E2 -1158.301} C_VEL
LIN {X 0,Y 594.59,Z 329.28,A -85,B 0,C 180,E1 -1158.746,E2 -1158.746} C_VEL
LIN {X 0,Y 594.536,Z 340.636,A -85,B 0,C 180,E1 -1159.27,E2 -1159.27} C_VEL
LIN {X 0,Y 594.477,Z 352.205,A -85,B 0,C 180,E1 -1159.958,E2 -1159.958} C_VEL
LIN {X 0,Y 594.414,Z 362.601,A -85,B 0,C 180,E1 -1160.73,E2 -1160.73} C_VEL
LIN {X 0,Y 594.383,Z 371.115,A -85,B 0,C 180,E1 -1161.501,E2 -1161.501} C_VEL
LIN {X 0,Y 594.347,Z 378.963,A -85,B 0,C 180,E1 -1162.356,E2 -1162.356} C_VEL
LIN {X 0,Y 594.282,Z 386.815,A -85,B 0,C 180,E1 -1163.409,E2 -1163.409} C_VEL
LIN {X 0,Y 594.289,Z 393.682,A -85,B 0,C 180,E1 -1164.572,E2 -1164.572} C_VEL
LIN {X 0,Y 594.27,Z 398.372,A -85,B 0,C 180,E1 -1165.592,E2 -1165.592} C_VEL
LIN {X 0,Y 594.267,Z 401.957,A -85,B 0,C 180,E1 -1166.61,E2 -1166.61} C_VEL
LIN {X 0,Y 594.226,Z 403.809,A -85,B 0,C 180,E1 -1167.289,E2 -1167.289} C_VEL
LIN {X 0,Y 594.242,Z 405.201,A -85,B 0,C 180,E1 -1167.967,E2 -1167.967} C_VEL
LIN {X 0,Y 594.239,Z 406.784,A -85,B 0,C 180,E1 -1169.323,E2 -1169.323} C_VEL
LIN {X 0,Y 594.236,Z 407,A -85,B 0,C 180,E1 -1170,E2 -1170} C_VEL
LIN {X 0,Y 594.247,Z 406.185,A -85,B 0,C 180,E1 -1171.356,E2 -1171.356} C_VEL
LIN {X 0,Y 594.242,Z 405.201,A -85,B 0,C 180,E1 -1172.034,E2 -1172.034} C_VEL
LIN {X 0,Y 594.226,Z 403.809,A -85,B 0,C 180,E1 -1172.712,E2 -1172.712} C_VEL
LIN {X 0,Y 594.289,Z 400.895,A -85,B 0,C 180,E1 -1173.73,E2 -1173.73} C_VEL
LIN {X 0,Y 594.241,Z 396.948,A -85,B 0,C 180,E1 -1174.749,E2 -1174.749} C_VEL
LIN {X 0,Y 594.305,Z 390.876,A -85,B 0,C 180,E1 -1175.939,E2 -1175.939} C_VEL
LIN {X 0,Y 594.308,Z 384.235,A -85,B 0,C 180,E1 -1176.962,E2 -1176.962} C_VEL
LIN {X 0,Y 594.359,Z 375.988,A -85,B 0,C 180,E1 -1177.987,E2 -1177.987} C_VEL
LIN {X 0,Y 594.382,Z 367.535,A -85,B 0,C 180,E1 -1178.842,E2 -1178.842} C_VEL
LIN {X 0,Y 594.432,Z 357.092,A -85,B 0,C 180,E1 -1179.7,E2 -1179.7} C_VEL
LIN {X 0,Y 594.482,Z 346.754,A -85,B 0,C 180,E1 -1180.387,E2 -1180.387} C_VEL
LIN {X 0,Y 594.558,Z 335.725,A -85,B 0,C 180,E1 -1180.973,E2 -1180.973} C_VEL
LIN {X 0,Y 594.579,Z 323.706,A -85,B 0,C 180,E1 -1181.464,E2 -1181.464} C_VEL
LIN {X 0,Y 594.648,Z 310.34,A -85,B 0,C 180,E1 -1181.85,E2 -1181.85} C_VEL
LIN {X 0,Y 594.697,Z 297.066,A -85,B 0,C 180,E1 -1182.087,E2 -1182.087} C_VEL
LIN {X 0,Y 594.623,Z 195.793,A -85,B 0,C 180,E1 -1183.317,E2 -1183.317} C_VEL
LIN {X 0,Y 594.429,Z 194.268,A -85,B 0,C 180,E1 -1183.351,E2 -1183.351} C_VEL
LIN {X 0,Y 594.529,Z 171.237,A -85,B 0,C 180,E1 -1186.305,E2 -1186.305} C_VEL
LIN {X 0,Y 594.613,Z 153.496,A -85,B 0,C 180,E1 -1188.61,E2 -1188.61} C_VEL
LIN {X 0,Y 594.746,Z 132.814,A -85,B 0,C 180,E1 -1191.335,E2 -1191.335} C_VEL
LIN {X 0,Y 594.821,Z 116.629,A -85,B 0,C 180,E1 -1193.501,E2 -1193.501} C_VEL
LIN {X 0,Y 594.392,Z 114.445,A -85,B 0,C 180,E1 -1193.82,E2 -1193.82} C_VEL
LIN {X 0,Y 594.385,Z 114.447,A -85,B 0,C 180,E1 -1196.7,E2 -1196.7} C_VEL
LIN {X 0,Y 594.385,Z 114.443,A -85,B 0,C 180,E1 -1198.999,E2 -1198.999} C_VEL
LIN {X 0,Y 594.381,Z 114.443,A -85,B 0,C 180,E1 -1201.643,E2 -1201.643} C_VEL
LIN {X 0,Y 594.379,Z 114.445,A -85,B 0,C 180,E1 -1204.58,E2 -1204.58} C_VEL
LIN {X 0,Y 594.394,Z 114.442,A -85,B 0,C 180,E1 -1207.609,E2 -1207.609} C_VEL
LIN {X 0,Y 594.372,Z 114.444,A -85,B 0,C 180,E1 -1210.567,E2 -1210.567} C_VEL
LIN {X 0,Y 594.37,Z 114.444,A -85,B 0,C 180,E1 -1213.299,E2 -1213.299} C_VEL
LIN {X 0,Y 594.372,Z 114.447,A -85,B 0,C 180,E1 -1216.16,E2 -1216.16} C_VEL
LIN {X 0,Y 594.381,Z 114.441,A -85,B 0,C 180,E1 -1218.536,E2 -1218.536} C_VEL
LIN {X 0,Y 594.385,Z 114.444,A -85,B 0,C 180,E1 -1221.296,E2 -1221.296} C_VEL
LIN {X 0,Y 594.353,Z 114.452,A -85,B 0,C 180,E1 -1223.755,E2 -1223.755} C_VEL
LIN {X 0,Y 594.367,Z 114.443,A -85,B 0,C 180,E1 -1226.238,E2 -1226.238} C_VEL
LIN {X 0,Y 594.371,Z 114.442,A -85,B 0,C 180,E1 -1228.65,E2 -1228.65} C_VEL
LIN {X 0,Y 594.386,Z 114.445,A -85,B 0,C 180,E1 -1231.042,E2 -1231.042} C_VEL
LIN {X 0,Y 594.38,Z 114.442,A -85,B 0,C 180,E1 -1233.979,E2 -1233.979} C_VEL
LIN {X 0,Y 594.371,Z 114.442,A -85,B 0,C 180,E1 -1236.295,E2 -1236.295} C_VEL
LIN {X 0,Y 594.4,Z 114.447,A -85,B 0,C 180,E1 -1239.224,E2 -1239.224} C_VEL
LIN {X 0,Y 594.343,Z 114.445,A -85,B 0,C 180,E1 -1242.094,E2 -1242.094} C_VEL
LIN {X 0,Y 594.362,Z 114.444,A -85,B 0,C 180,E1 -1244.219,E2 -1244.219} C_VEL
LIN {X 0,Y 594.358,Z 114.452,A -85,B 0,C 180,E1 -1247.017,E2 -1247.017} C_VEL
LIN {X 0,Y 594.386,Z 114.44,A -85,B 0,C 180,E1 -1249.784,E2 -1249.784} C_VEL
LIN {X 0,Y 594.394,Z 114.446,A -85,B 0,C 180,E1 -1252.527,E2 -1252.527} C_VEL
LIN {X 0,Y 594.371,Z 114.444,A -85,B 0,C 180,E1 -1255.252,E2 -1255.252} C_VEL
LIN {X 0,Y 594.404,Z 114.44,A -85,B 0,C 180,E1 -1257.967,E2 -1257.967} C_VEL
LIN {X 0,Y 594.413,Z 114.444,A -85,B 0,C 180,E1 -1260.677,E2 -1260.677} C_VEL
LIN {X 0,Y 594.396,Z 114.445,A -85,B 0,C 180,E1 -1262.711,E2 -1262.711} C_VEL
LIN {X 0,Y 594.374,Z 114.442,A -85,B 0,C 180,E1 -1265.428,E2 -1265.428} C_VEL
LIN {X 0,Y 594.397,Z 114.478,A -85,B 0,C 180,E1 -1267.558,E2 -1267.558} C_VEL
LIN {X 0,Y 594.371,Z 130.55,A -85,B 0,C 180,E1 -1270.56,E2 -1270.56} C_VEL
LIN {X 0,Y 594.387,Z 136.844,A -85,B 0,C 180,E1 -1271.725,E2 -1271.725} C_VEL
LIN {X 0,Y 594.783,Z 143.522,A -85,B 0,C 180,E1 -1271.825,E2 -1271.825} C_VEL
LIN {X 0,Y 594.737,Z 159.793,A -85,B 0,C 180,E1 -1272.022,E2 -1272.022} C_VEL
LIN {X 0,Y 594.048,Z 165.634,A -85,B 0,C 180,E1 -1272.078,E2 -1272.078} C_VEL
LIN {X 0,Y 588.509,Z 184.637,A -85,B 0,C 180,E1 -1272.187,E2 -1272.187} C_VEL
LIN {X 0,Y 587.823,Z 190.478,A -85,B 0,C 180,E1 -1272.243,E2 -1272.243} C_VEL
LIN {X 0,Y 587.716,Z 243.656,A -85,B 0,C 180,E1 -1272.913,E2 -1272.913} C_VEL
LIN {X 0,Y 587.672,Z 256.687,A -85,B 0,C 180,E1 -1273.221,E2 -1273.221} C_VEL
LIN {X 0,Y 587.605,Z 269.463,A -85,B 0,C 180,E1 -1273.663,E2 -1273.663} C_VEL
LIN {X 0,Y 587.487,Z 282.106,A -85,B 0,C 180,E1 -1274.267,E2 -1274.267} C_VEL
LIN {X 0,Y 587.445,Z 292.508,A -85,B 0,C 180,E1 -1274.905,E2 -1274.905} C_VEL
LIN {X 0,Y 587.352,Z 302.007,A -85,B 0,C 180,E1 -1275.618,E2 -1275.618} C_VEL
LIN {X 0,Y 587.318,Z 311.778,A -85,B 0,C 180,E1 -1276.511,E2 -1276.511} C_VEL
LIN {X 0,Y 587.238,Z 321.196,A -85,B 0,C 180,E1 -1277.589,E2 -1277.589} C_VEL
LIN {X 0,Y 587.206,Z 328.704,A -85,B 0,C 180,E1 -1278.672,E2 -1278.672} C_VEL
LIN {X 0,Y 587.192,Z 333.808,A -85,B 0,C 180,E1 -1279.58,E2 -1279.58} C_VEL
LIN {X 0,Y 587.165,Z 338.631,A -85,B 0,C 180,E1 -1280.654,E2 -1280.654} C_VEL
LIN {X 0,Y 587.174,Z 342.442,A -85,B 0,C 180,E1 -1281.78,E2 -1281.78} C_VEL
LIN {X 0,Y 587.127,Z 344.902,A -85,B 0,C 180,E1 -1282.824,E2 -1282.824} C_VEL
LIN {X 0,Y 587.125,Z 346.553,A -85,B 0,C 180,E1 -1284.015,E2 -1284.015} C_VEL
LIN {X 0,Y 587.133,Z 346.943,A -85,B 0,C 180,E1 -1284.768,E2 -1284.768} C_VEL
LIN {X 0,Y 587.12,Z 346.5,A -85,B 0,C 180,E1 -1286.133,E2 -1286.133} C_VEL
LIN {X 0,Y 587.131,Z 345.282,A -85,B 0,C 180,E1 -1287.056,E2 -1287.056} C_VEL
LIN {X 0,Y 587.152,Z 342.718,A -85,B 0,C 180,E1 -1288.216,E2 -1288.216} C_VEL
LIN {X 0,Y 587.194,Z 338.828,A -85,B 0,C 180,E1 -1289.388,E2 -1289.388} C_VEL
LIN {X 0,Y 587.193,Z 333.932,A -85,B 0,C 180,E1 -1290.486,E2 -1290.486} C_VEL
LIN {X 0,Y 587.235,Z 327.74,A -85,B 0,C 180,E1 -1291.574,E2 -1291.574} C_VEL
LIN {X 0,Y 587.251,Z 320.542,A -85,B 0,C 180,E1 -1292.584,E2 -1292.584} C_VEL
LIN {X 0,Y 587.336,Z 311.545,A -85,B 0,C 180,E1 -1293.602,E2 -1293.602} C_VEL
LIN {X 0,Y 587.404,Z 302.124,A -85,B 0,C 180,E1 -1294.462,E2 -1294.462} C_VEL
LIN {X 0,Y 587.458,Z 291.927,A -85,B 0,C 180,E1 -1295.225,E2 -1295.225} C_VEL
LIN {X 0,Y 587.53,Z 280.044,A -85,B 0,C 180,E1 -1295.936,E2 -1295.936} C_VEL
LIN {X 0,Y 587.615,Z 267.228,A -85,B 0,C 180,E1 -1296.514,E2 -1296.514} C_VEL
LIN {X 0,Y 587.612,Z 255.86,A -85,B 0,C 180,E1 -1296.893,E2 -1296.893} C_VEL
LIN {X 0,Y 587.722,Z 243.088,A -85,B 0,C 180,E1 -1297.188,E2 -1297.188} C_VEL
LIN {X 0,Y 587.7,Z 139.528,A -85,B 0,C 180,E1 -1298.476,E2 -1298.476} C_VEL
LIN {X 0,Y 587.293,Z 136.797,A -85,B 0,C 180,E1 -1298.537,E2 -1298.537} C_VEL
LIN {X 0,Y 587.382,Z 122.874,A -85,B 0,C 180,E1 -1301.153,E2 -1301.153} C_VEL
LIN {X 0,Y 587.367,Z 115.318,A -85,B 0,C 180,E1 -1302.592,E2 -1302.592} C_VEL
LIN {X 0,Y 587.317,Z 115.322,A -85,B 0,C 180,E1 -1305.088,E2 -1305.088} C_VEL
LIN {X 0,Y 587.354,Z 115.323,A -85,B 0,C 180,E1 -1307.927,E2 -1307.927} C_VEL
LIN {X 0,Y 587.324,Z 115.321,A -85,B 0,C 180,E1 -1311.059,E2 -1311.059} C_VEL
LIN {X 0,Y 587.348,Z 115.322,A -85,B 0,C 180,E1 -1313.292,E2 -1313.292} C_VEL
LIN {X 0,Y 587.334,Z 115.325,A -85,B 0,C 180,E1 -1315.778,E2 -1315.778} C_VEL
LIN {X 0,Y 587.341,Z 115.318,A -85,B 0,C 180,E1 -1318.231,E2 -1318.231} C_VEL
LIN {X 0,Y 587.348,Z 115.318,A -85,B 0,C 180,E1 -1320.866,E2 -1320.866} C_VEL
LIN {X 0,Y 587.357,Z 115.319,A -85,B 0,C 180,E1 -1323.819,E2 -1323.819} C_VEL
LIN {X 0,Y 587.324,Z 115.321,A -85,B 0,C 180,E1 -1325.993,E2 -1325.993} C_VEL
LIN {X 0,Y 587.32,Z 115.32,A -85,B 0,C 180,E1 -1328.225,E2 -1328.225} C_VEL
LIN {X 0,Y 587.347,Z 115.326,A -85,B 0,C 180,E1 -1331.151,E2 -1331.151} C_VEL
LIN {X 0,Y 587.319,Z 115.32,A -85,B 0,C 180,E1 -1334.024,E2 -1334.024} C_VEL
LIN {X 0,Y 587.359,Z 115.315,A -85,B 0,C 180,E1 -1336.154,E2 -1336.154} C_VEL
LIN {X 0,Y 587.338,Z 115.327,A -85,B 0,C 180,E1 -1338.962,E2 -1338.962} C_VEL
LIN {X 0,Y 587.362,Z 115.315,A -85,B 0,C 180,E1 -1341.744,E2 -1341.744} C_VEL
LIN {X 0,Y 587.365,Z 115.318,A -85,B 0,C 180,E1 -1344.507,E2 -1344.507} C_VEL
LIN {X 0,Y 587.365,Z 115.318,A -85,B 0,C 180,E1 -1347.256,E2 -1347.256} C_VEL
LIN {X 0,Y 587.383,Z 115.313,A -85,B 0,C 180,E1 -1350,E2 -1350} C_VEL
LIN {X 0,Y 587.373,Z 115.324,A -85,B 0,C 180,E1 -1352.743,E2 -1352.743} C_VEL
LIN {X 0,Y 587.356,Z 115.316,A -85,B 0,C 180,E1 -1355.493,E2 -1355.493} C_VEL
LIN {X 0,Y 587.371,Z 115.318,A -85,B 0,C 180,E1 -1358.255,E2 -1358.255} C_VEL
LIN {X 0,Y 587.347,Z 115.319,A -85,B 0,C 180,E1 -1361.133,E2 -1361.133} C_VEL
LIN {X 0,Y 587.363,Z 115.321,A -85,B 0,C 180,E1 -1364.26,E2 -1364.26} C_VEL
LIN {X 0,Y 587.347,Z 115.317,A -85,B 0,C 180,E1 -1367.406,E2 -1367.406} C_VEL
LIN {X 0,Y 587.328,Z 115.328,A -85,B 0,C 180,E1 -1370.305,E2 -1370.305} C_VEL
LIN {X 0,Y 587.313,Z 115.321,A -85,B 0,C 180,E1 -1373.259,E2 -1373.259} C_VEL
LIN {X 0,Y 587.333,Z 115.319,A -85,B 0,C 180,E1 -1375.516,E2 -1375.516} C_VEL
LIN {X 0,Y 587.344,Z 115.321,A -85,B 0,C 180,E1 -1377.818,E2 -1377.818} C_VEL
LIN {X 0,Y 587.349,Z 115.321,A -85,B 0,C 180,E1 -1380.512,E2 -1380.512} C_VEL
LIN {X 0,Y 587.333,Z 115.319,A -85,B 0,C 180,E1 -1383.396,E2 -1383.396} C_VEL
LIN {X 0,Y 587.343,Z 115.325,A -85,B 0,C 180,E1 -1385.896,E2 -1385.896} C_VEL
LIN {X 0,Y 587.331,Z 115.321,A -85,B 0,C 180,E1 -1388.479,E2 -1388.479} C_VEL
LIN {X 0,Y 587.334,Z 115.319,A -85,B 0,C 180,E1 -1391.157,E2 -1391.157} C_VEL
LIN {X 0,Y 587.332,Z 115.325,A -85,B 0,C 180,E1 -1394.114,E2 -1394.114} C_VEL
LIN {X 0,Y 587.314,Z 115.321,A -85,B 0,C 180,E1 -1396.994,E2 -1396.994} C_VEL
LIN {X 0,Y 587.316,Z 115.331,A -85,B 0,C 180,E1 -1399.746,E2 -1399.746} C_VEL
LIN {X 0,Y 587.343,Z 115.318,A -85,B 0,C 180,E1 -1402.393,E2 -1402.393} C_VEL
LIN {X 0,Y 587.359,Z 115.323,A -85,B 0,C 180,E1 -1405.78,E2 -1405.78} C_VEL
LIN {X 0,Y 587.351,Z 115.317,A -85,B 0,C 180,E1 -1408.232,E2 -1408.232} C_VEL
LIN {X 0,Y 587.347,Z 115.318,A -85,B 0,C 180,E1 -1410.867,E2 -1410.867} C_VEL
LIN {X 0,Y 587.356,Z 115.32,A -85,B 0,C 180,E1 -1413.819,E2 -1413.819} C_VEL
LIN {X 0,Y 587.332,Z 115.32,A -85,B 0,C 180,E1 -1415.994,E2 -1415.994} C_VEL
LIN {X 0,Y 587.322,Z 115.32,A -85,B 0,C 180,E1 -1418.226,E2 -1418.226} C_VEL
LIN {X 0,Y 587.348,Z 115.325,A -85,B 0,C 180,E1 -1421.151,E2 -1421.151} C_VEL
LIN {X 0,Y 587.32,Z 115.32,A -85,B 0,C 180,E1 -1424.025,E2 -1424.025} C_VEL
LIN {X 0,Y 587.358,Z 115.315,A -85,B 0,C 180,E1 -1426.155,E2 -1426.155} C_VEL
LIN {X 0,Y 587.339,Z 115.325,A -85,B 0,C 180,E1 -1428.963,E2 -1428.963} C_VEL
LIN {X 0,Y 587.362,Z 115.316,A -85,B 0,C 180,E1 -1431.745,E2 -1431.745} C_VEL
LIN {X 0,Y 587.363,Z 115.318,A -85,B 0,C 180,E1 -1434.507,E2 -1434.507} C_VEL
LIN {X 0,Y 587.367,Z 115.319,A -85,B 0,C 180,E1 -1437.257,E2 -1437.257} C_VEL
LIN {X 0,Y 587.383,Z 115.312,A -85,B 0,C 180,E1 -1440,E2 -1440} C_VEL
LIN {X 0,Y 587.37,Z 115.323,A -85,B 0,C 180,E1 -1442.744,E2 -1442.744} C_VEL
LIN {X 0,Y 587.358,Z 115.316,A -85,B 0,C 180,E1 -1445.493,E2 -1445.493} C_VEL
LIN {X 0,Y 587.37,Z 115.317,A -85,B 0,C 180,E1 -1448.255,E2 -1448.255} C_VEL
LIN {X 0,Y 587.347,Z 115.319,A -85,B 0,C 180,E1 -1451.134,E2 -1451.134} C_VEL
LIN {X 0,Y 587.364,Z 115.32,A -85,B 0,C 180,E1 -1454.261,E2 -1454.261} C_VEL
LIN {X 0,Y 587.348,Z 115.317,A -85,B 0,C 180,E1 -1457.406,E2 -1457.406} C_VEL
LIN {X 0,Y 587.329,Z 115.327,A -85,B 0,C 180,E1 -1460.305,E2 -1460.305} C_VEL
LIN {X 0,Y 587.313,Z 115.321,A -85,B 0,C 180,E1 -1463.259,E2 -1463.259} C_VEL
LIN {X 0,Y 587.334,Z 115.319,A -85,B 0,C 180,E1 -1465.517,E2 -1465.517} C_VEL
LIN {X 0,Y 587.346,Z 115.32,A -85,B 0,C 180,E1 -1467.818,E2 -1467.818} C_VEL
LIN {X 0,Y 587.336,Z 115.323,A -85,B 0,C 180,E1 -1470.51,E2 -1470.51} C_VEL
LIN {X 0,Y 587.334,Z 115.319,A -85,B 0,C 180,E1 -1473.397,E2 -1473.397} C_VEL
LIN {X 0,Y 587.29,Z 115.331,A -85,B 0,C 180,E1 -1475.9,E2 -1475.9} C_VEL
LIN {X 0,Y 587.333,Z 115.322,A -85,B 0,C 180,E1 -1478.479,E2 -1478.479} C_VEL
LIN {X 0,Y 587.337,Z 115.318,A -85,B 0,C 180,E1 -1481.157,E2 -1481.157} C_VEL
LIN {X 0,Y 587.327,Z 115.326,A -85,B 0,C 180,E1 -1484.114,E2 -1484.114} C_VEL
LIN {X 0,Y 587.315,Z 115.321,A -85,B 0,C 180,E1 -1486.994,E2 -1486.994} C_VEL
LIN {X 0,Y 587.319,Z 115.33,A -85,B 0,C 180,E1 -1489.746,E2 -1489.746} C_VEL
LIN {X 0,Y 587.346,Z 115.318,A -85,B 0,C 180,E1 -1492.393,E2 -1492.393} C_VEL
LIN {X 0,Y 587.361,Z 115.323,A -85,B 0,C 180,E1 -1495.78,E2 -1495.78} C_VEL
LIN {X 0,Y 587.343,Z 115.319,A -85,B 0,C 180,E1 -1498.232,E2 -1498.232} C_VEL
LIN {X 0,Y 587.351,Z 115.317,A -85,B 0,C 180,E1 -1500.867,E2 -1500.867} C_VEL
LIN {X 0,Y 587.36,Z 115.322,A -85,B 0,C 180,E1 -1503.82,E2 -1503.82} C_VEL
LIN {X 0,Y 587.384,Z 115.452,A -85,B 0,C 180,E1 -1506.066,E2 -1506.066} C_VEL
LIN {X 0,Y 587.927,Z 119.134,A -85,B 0,C 180,E1 -1506.58,E2 -1506.58} C_VEL
LIN {X 0,Y 587.784,Z 138.488,A -85,B 0,C 180,E1 -1509.163,E2 -1509.163} C_VEL
LIN {X 0,Y 587.678,Z 158.959,A -85,B 0,C 180,E1 -1511.885,E2 -1511.885} C_VEL
LIN {X 0,Y 587.5,Z 180.795,A -85,B 0,C 180,E1 -1514.742,E2 -1514.742} C_VEL
LIN {X 0,Y 587.386,Z 194.357,A -85,B 0,C 180,E1 -1516.497,E2 -1516.497} C_VEL
LIN {X 0,Y 587.862,Z 200.531,A -85,B 0,C 180,E1 -1516.585,E2 -1516.585} C_VEL
LIN {X 0,Y 587.726,Z 302.961,A -85,B 0,C 180,E1 -1517.855,E2 -1517.855} C_VEL
LIN {X 0,Y 587.655,Z 316.229,A -85,B 0,C 180,E1 -1518.16,E2 -1518.16} C_VEL
LIN {X 0,Y 587.619,Z 328.975,A -85,B 0,C 180,E1 -1518.599,E2 -1518.599} C_VEL
LIN {X 0,Y 587.557,Z 340.634,A -85,B 0,C 180,E1 -1519.141,E2 -1519.141} C_VEL
LIN {X 0,Y 587.464,Z 352.207,A -85,B 0,C 180,E1 -1519.837,E2 -1519.837} C_VEL
LIN {X 0,Y 587.394,Z 362.602,A -85,B 0,C 180,E1 -1520.618,E2 -1520.618} C_VEL
LIN {X 0,Y 587.321,Z 371.115,A -85,B 0,C 180,E1 -1521.398,E2 -1521.398} C_VEL
LIN {X 0,Y 587.274,Z 378.963,A -85,B 0,C 180,E1 -1522.263,E2 -1522.263} C_VEL
LIN {X 0,Y 587.23,Z 385.471,A -85,B 0,C 180,E1 -1523.127,E2 -1523.127} C_VEL
LIN {X 0,Y 587.237,Z 391.868,A -85,B 0,C 180,E1 -1524.162,E2 -1524.162} C_VEL
LIN {X 0,Y 587.147,Z 396.951,A -85,B 0,C 180,E1 -1525.194,E2 -1525.194} C_VEL
LIN {X 0,Y 587.213,Z 400.896,A -85,B 0,C 180,E1 -1526.226,E2 -1526.226} C_VEL
LIN {X 0,Y 587.132,Z 403.809,A -85,B 0,C 180,E1 -1527.256,E2 -1527.256} C_VEL
LIN {X 0,Y 587.141,Z 405.2,A -85,B 0,C 180,E1 -1527.942,E2 -1527.942} C_VEL
LIN {X 0,Y 587.14,Z 406.785,A -85,B 0,C 180,E1 -1529.314,E2 -1529.314} C_VEL
LIN {X 0,Y 587.137,Z 407,A -85,B 0,C 180,E1 -1530,E2 -1530} C_VEL
LIN {X 0,Y 587.147,Z 406.185,A -85,B 0,C 180,E1 -1531.372,E2 -1531.372} C_VEL
LIN {X 0,Y 587.141,Z 405.2,A -85,B 0,C 180,E1 -1532.058,E2 -1532.058} C_VEL
LIN {X 0,Y 587.132,Z 403.809,A -85,B 0,C 180,E1 -1532.745,E2 -1532.745} C_VEL
LIN {X 0,Y 587.213,Z 400.895,A -85,B 0,C 180,E1 -1533.775,E2 -1533.775} C_VEL
LIN {X 0,Y 587.147,Z 396.948,A -85,B 0,C 180,E1 -1534.807,E2 -1534.807} C_VEL
LIN {X 0,Y 587.218,Z 390.876,A -85,B 0,C 180,E1 -1536.011,E2 -1536.011} C_VEL
LIN {X 0,Y 587.245,Z 384.235,A -85,B 0,C 180,E1 -1537.046,E2 -1537.046} C_VEL
LIN {X 0,Y 587.3,Z 375.988,A -85,B 0,C 180,E1 -1538.083,E2 -1538.083} C_VEL
LIN {X 0,Y 587.343,Z 367.535,A -85,B 0,C 180,E1 -1538.949,E2 -1538.949} C_VEL
LIN {X 0,Y 587.419,Z 357.093,A -85,B 0,C 180,E1 -1539.817,E2 -1539.817} C_VEL
LIN {X 0,Y 587.497,Z 346.752,A -85,B 0,C 180,E1 -1540.512,E2 -1540.512} C_VEL
LIN {X 0,Y 587.561,Z 334.814,A -85,B 0,C 180,E1 -1541.149,E2 -1541.149} C_VEL
LIN {X 0,Y 587.629,Z 322.592,A -85,B 0,C 180,E1 -1541.639,E2 -1541.639} C_VEL
LIN {X 0,Y 587.703,Z 309.424,A -85,B 0,C 180,E1 -1542.014,E2 -1542.014} C_VEL
LIN {X 0,Y 587.769,Z 297.066,A -85,B 0,C 180,E1 -1542.232,E2 -1542.232} C_VEL
LIN {X 0,Y 587.714,Z 196.464,A -85,B 0,C 180,E1 -1543.468,E2 -1543.468} C_VEL
LIN {X 0,Y 587.394,Z 194.268,A -85,B 0,C 180,E1 -1543.514,E2 -1543.514} C_VEL
LIN {X 0,Y 587.551,Z 172.602,A -85,B 0,C 180,E1 -1546.326,E2 -1546.326} C_VEL
LIN {X 0,Y 587.641,Z 153.496,A -85,B 0,C 180,E1 -1548.839,E2 -1548.839} C_VEL
LIN {X 0,Y 587.832,Z 134.341,A -85,B 0,C 180,E1 -1551.393,E2 -1551.393} C_VEL
LIN {X 0,Y 587.931,Z 118.949,A -85,B 0,C 180,E1 -1553.42,E2 -1553.42} C_VEL
LIN {X 0,Y 587.353,Z 115.323,A -85,B 0,C 180,E1 -1553.936,E2 -1553.936} C_VEL
LIN {X 0,Y 587.342,Z 115.326,A -85,B 0,C 180,E1 -1556.279,E2 -1556.279} C_VEL
LIN {X 0,Y 587.353,Z 115.318,A -85,B 0,C 180,E1 -1559.133,E2 -1559.133} C_VEL
LIN {X 0,Y 587.348,Z 115.321,A -85,B 0,C 180,E1 -1561.836,E2 -1561.836} C_VEL
LIN {X 0,Y 587.349,Z 115.325,A -85,B 0,C 180,E1 -1564.347,E2 -1564.347} C_VEL
LIN {X 0,Y 587.349,Z 115.32,A -85,B 0,C 180,E1 -1567.608,E2 -1567.608} C_VEL
LIN {X 0,Y 587.316,Z 115.327,A -85,B 0,C 180,E1 -1570.254,E2 -1570.254} C_VEL
LIN {X 0,Y 587.318,Z 115.321,A -85,B 0,C 180,E1 -1573.118,E2 -1573.118} C_VEL
LIN {X 0,Y 587.327,Z 115.326,A -85,B 0,C 180,E1 -1576.05,E2 -1576.05} C_VEL
LIN {X 0,Y 587.339,Z 115.318,A -85,B 0,C 180,E1 -1578.925,E2 -1578.925} C_VEL
LIN {X 0,Y 587.331,Z 115.326,A -85,B 0,C 180,E1 -1581.52,E2 -1581.52} C_VEL
LIN {X 0,Y 587.293,Z 115.326,A -85,B 0,C 180,E1 -1584.1,E2 -1584.1} C_VEL
LIN {X 0,Y 587.34,Z 115.319,A -85,B 0,C 180,E1 -1586.888,E2 -1586.888} C_VEL
LIN {X 0,Y 587.329,Z 115.329,A -85,B 0,C 180,E1 -1589.492,E2 -1589.492} C_VEL
LIN {X 0,Y 587.345,Z 115.317,A -85,B 0,C 180,E1 -1592.309,E2 -1592.309} C_VEL
LIN {X 0,Y 587.353,Z 115.326,A -85,B 0,C 180,E1 -1595.241,E2 -1595.241} C_VEL
LIN {X 0,Y 587.318,Z 115.321,A -85,B 0,C 180,E1 -1598.225,E2 -1598.225} C_VEL
LIN {X 0,Y 587.346,Z 115.326,A -85,B 0,C 180,E1 -1601.151,E2 -1601.151} C_VEL
LIN {X 0,Y 587.315,Z 115.321,A -85,B 0,C 180,E1 -1604.024,E2 -1604.024} C_VEL
LIN {X 0,Y 587.353,Z 115.317,A -85,B 0,C 180,E1 -1606.154,E2 -1606.154} C_VEL
LIN {X 0,Y 587.34,Z 115.326,A -85,B 0,C 180,E1 -1608.962,E2 -1608.962} C_VEL
LIN {X 0,Y 587.34,Z 115.318,A -85,B 0,C 180,E1 -1611.744,E2 -1611.744} C_VEL
LIN {X 0,Y 587.365,Z 115.323,A -85,B 0,C 180,E1 -1614.507,E2 -1614.507} C_VEL
LIN {X 0,Y 587.355,Z 115.318,A -85,B 0,C 180,E1 -1617.256,E2 -1617.256} C_VEL
LIN {X 0,Y 587.384,Z 115.315,A -85,B 0,C 180,E1 -1620,E2 -1620} C_VEL
LIN {X 0,Y 587.361,Z 115.321,A -85,B 0,C 180,E1 -1622.743,E2 -1622.743} C_VEL
LIN {X 0,Y 587.344,Z 115.319,A -85,B 0,C 180,E1 -1625.493,E2 -1625.493} C_VEL
LIN {X 0,Y 587.366,Z 115.409,A -85,B 0,C 180,E1 -1627.52,E2 -1627.52} C_VEL
LIN {X 0,Y 587.323,Z 128.47,A -85,B 0,C 180,E1 -1629.992,E2 -1629.992} C_VEL
LIN {X 0,Y 587.333,Z 136.853,A -85,B 0,C 180,E1 -1631.564,E2 -1631.564} C_VEL
LIN {X 0,Y 587.865,Z 141.842,A -85,B 0,C 180,E1 -1631.646,E2 -1631.646} C_VEL
LIN {X 0,Y 587.823,Z 190.478,A -85,B 0,C 180,E1 -1632.243,E2 -1632.243} C_VEL
LIN {X 0,Y 587.117,Z 196.322,A -85,B 0,C 180,E1 -1632.299,E2 -1632.299} C_VEL
LIN {X 0,Y 581.479,Z 215.312,A -85,B 0,C 180,E1 -1632.409,E2 -1632.409} C_VEL
LIN {X 0,Y 580.833,Z 221.154,A -85,B 0,C 180,E1 -1632.467,E2 -1632.467} C_VEL
LIN {X 0,Y 580.787,Z 244.428,A -85,B 0,C 180,E1 -1632.78,E2 -1632.78} C_VEL
LIN {X 0,Y 580.715,Z 256.418,A -85,B 0,C 180,E1 -1633.071,E2 -1633.071} C_VEL
LIN {X 0,Y 580.639,Z 268.159,A -85,B 0,C 180,E1 -1633.473,E2 -1633.473} C_VEL
LIN {X 0,Y 580.523,Z 281.434,A -85,B 0,C 180,E1 -1634.098,E2 -1634.098} C_VEL
LIN {X 0,Y 580.415,Z 291.775,A -85,B 0,C 180,E1 -1634.731,E2 -1634.731} C_VEL
LIN {X 0,Y 580.311,Z 301.387,A -85,B 0,C 180,E1 -1635.452,E2 -1635.452} C_VEL
LIN {X 0,Y 580.314,Z 309.395,A -85,B 0,C 180,E1 -1636.173,E2 -1636.173} C_VEL
LIN {X 0,Y 580.209,Z 317.825,A -85,B 0,C 180,E1 -1637.082,E2 -1637.082} C_VEL
LIN {X 0,Y 580.16,Z 326.069,A -85,B 0,C 180,E1 -1638.175,E2 -1638.175} C_VEL
LIN {X 0,Y 580.156,Z 331.73,A -85,B 0,C 180,E1 -1639.11,E2 -1639.11} C_VEL
LIN {X 0,Y 580.107,Z 337.006,A -85,B 0,C 180,E1 -1640.198,E2 -1640.198} C_VEL
LIN {X 0,Y 580.069,Z 341.137,A -85,B 0,C 180,E1 -1641.313,E2 -1641.313} C_VEL
LIN {X 0,Y 580.056,Z 343.3,A -85,B 0,C 180,E1 -1642.061,E2 -1642.061} C_VEL
LIN {X 0,Y 580.045,Z 345.192,A -85,B 0,C 180,E1 -1642.951,E2 -1642.951} C_VEL
LIN {X 0,Y 580.028,Z 346.761,A -85,B 0,C 180,E1 -1644.328,E2 -1644.328} C_VEL
LIN {X 0,Y 580.024,Z 346.995,A -85,B 0,C 180,E1 -1645.093,E2 -1645.093} C_VEL
LIN {X 0,Y 580.047,Z 346.345,A -85,B 0,C 180,E1 -1646.284,E2 -1646.284} C_VEL
LIN {X 0,Y 580.06,Z 343.795,A -85,B 0,C 180,E1 -1647.814,E2 -1647.814} C_VEL
LIN {X 0,Y 580.08,Z 340.487,A -85,B 0,C 180,E1 -1648.987,E2 -1648.987} C_VEL
LIN {X 0,Y 580.093,Z 335.72,A -85,B 0,C 180,E1 -1650.184,E2 -1650.184} C_VEL
LIN {X 0,Y 580.128,Z 330.483,A -85,B 0,C 180,E1 -1651.198,E2 -1651.198} C_VEL
LIN {X 0,Y 580.182,Z 324.004,A -85,B 0,C 180,E1 -1652.207,E2 -1652.207} C_VEL
LIN {X 0,Y 580.223,Z 316.448,A -85,B 0,C 180,E1 -1653.168,E2 -1653.168} C_VEL
LIN {X 0,Y 580.333,Z 307.908,A -85,B 0,C 180,E1 -1654.062,E2 -1654.062} C_VEL
LIN {X 0,Y 580.384,Z 298.18,A -85,B 0,C 180,E1 -1654.901,E2 -1654.901} C_VEL
LIN {X 0,Y 580.5,Z 287.676,A -85,B 0,C 180,E1 -1655.628,E2 -1655.628} C_VEL
LIN {X 0,Y 580.554,Z 277.41,A -85,B 0,C 180,E1 -1656.201,E2 -1656.201} C_VEL
LIN {X 0,Y 580.632,Z 266.528,A -85,B 0,C 180,E1 -1656.679,E2 -1656.679} C_VEL
LIN {X 0,Y 580.698,Z 255.197,A -85,B 0,C 180,E1 -1657.054,E2 -1657.054} C_VEL
LIN {X 0,Y 580.765,Z 242.693,A -85,B 0,C 180,E1 -1657.342,E2 -1657.342} C_VEL
LIN {X 0,Y 580.894,Z 140.793,A -85,B 0,C 180,E1 -1658.621,E2 -1658.621} C_VEL
LIN {X 0,Y 580.257,Z 136.849,A -85,B 0,C 180,E1 -1658.694,E2 -1658.694} C_VEL
LIN {X 0,Y 580.353,Z 122.007,A -85,B 0,C 180,E1 -1661.519,E2 -1661.519} C_VEL
LIN {X 0,Y 580.311,Z 116.197,A -85,B 0,C 180,E1 -1662.656,E2 -1662.656} C_VEL
LIN {X 0,Y 580.27,Z 116.207,A -85,B 0,C 180,E1 -1665.609,E2 -1665.609} C_VEL
LIN {X 0,Y 580.299,Z 116.197,A -85,B 0,C 180,E1 -1668.233,E2 -1668.233} C_VEL
LIN {X 0,Y 580.278,Z 116.198,A -85,B 0,C 180,E1 -1670.965,E2 -1670.965} C_VEL
LIN {X 0,Y 580.268,Z 116.209,A -85,B 0,C 180,E1 -1673.596,E2 -1673.596} C_VEL
LIN {X 0,Y 580.3,Z 116.196,A -85,B 0,C 180,E1 -1676.144,E2 -1676.144} C_VEL
LIN {X 0,Y 580.274,Z 116.198,A -85,B 0,C 180,E1 -1678.614,E2 -1678.614} C_VEL
LIN {X 0,Y 580.291,Z 116.199,A -85,B 0,C 180,E1 -1681.024,E2 -1681.024} C_VEL
LIN {X 0,Y 580.29,Z 116.201,A -85,B 0,C 180,E1 -1683.666,E2 -1683.666} C_VEL
LIN {X 0,Y 580.295,Z 116.2,A -85,B 0,C 180,E1 -1685.683,E2 -1685.683} C_VEL
LIN {X 0,Y 580.271,Z 116.199,A -85,B 0,C 180,E1 -1687.947,E2 -1687.947} C_VEL
LIN {X 0,Y 580.298,Z 116.2,A -85,B 0,C 180,E1 -1690.913,E2 -1690.913} C_VEL
LIN {X 0,Y 580.274,Z 116.199,A -85,B 0,C 180,E1 -1693.825,E2 -1693.825} C_VEL
LIN {X 0,Y 580.326,Z 116.192,A -85,B 0,C 180,E1 -1695.983,E2 -1695.983} C_VEL
LIN {X 0,Y 580.304,Z 116.2,A -85,B 0,C 180,E1 -1698.827,E2 -1698.827} C_VEL
LIN {X 0,Y 580.326,Z 116.193,A -85,B 0,C 180,E1 -1701.644,E2 -1701.644} C_VEL
LIN {X 0,Y 580.331,Z 116.193,A -85,B 0,C 180,E1 -1704.44,E2 -1704.44} C_VEL
LIN {X 0,Y 580.333,Z 116.195,A -85,B 0,C 180,E1 -1707.223,E2 -1707.223} C_VEL
LIN {X 0,Y 580.352,Z 116.188,A -85,B 0,C 180,E1 -1710,E2 -1710} C_VEL
LIN {X 0,Y 580.339,Z 116.2,A -85,B 0,C 180,E1 -1712.776,E2 -1712.776} C_VEL
LIN {X 0,Y 580.324,Z 116.192,A -85,B 0,C 180,E1 -1715.559,E2 -1715.559} C_VEL
LIN {X 0,Y 580.334,Z 116.196,A -85,B 0,C 180,E1 -1718.356,E2 -1718.356} C_VEL
LIN {X 0,Y 580.299,Z 116.196,A -85,B 0,C 180,E1 -1721.191,E2 -1721.191} C_VEL
LIN {X 0,Y 580.323,Z 116.194,A -85,B 0,C 180,E1 -1724.017,E2 -1724.017} C_VEL
LIN {X 0,Y 580.31,Z 116.196,A -85,B 0,C 180,E1 -1726.914,E2 -1726.914} C_VEL
LIN {X 0,Y 580.303,Z 116.196,A -85,B 0,C 180,E1 -1729.822,E2 -1729.822} C_VEL
LIN {X 0,Y 580.289,Z 116.199,A -85,B 0,C 180,E1 -1732.802,E2 -1732.802} C_VEL
LIN {X 0,Y 580.305,Z 116.194,A -85,B 0,C 180,E1 -1735.079,E2 -1735.079} C_VEL
LIN {X 0,Y 580.296,Z 116.205,A -85,B 0,C 180,E1 -1738.185,E2 -1738.185} C_VEL
LIN {X 0,Y 580.296,Z 116.197,A -85,B 0,C 180,E1 -1740.697,E2 -1740.697} C_VEL
LIN {X 0,Y 580.302,Z 116.195,A -85,B 0,C 180,E1 -1743.316,E2 -1743.316} C_VEL
LIN {X 0,Y 580.29,Z 116.2,A -85,B 0,C 180,E1 -1746.402,E2 -1746.402} C_VEL
LIN {X 0,Y 580.306,Z 116.194,A -85,B 0,C 180,E1 -1749.187,E2 -1749.187} C_VEL
LIN {X 0,Y 580.311,Z 116.201,A -85,B 0,C 180,E1 -1751.766,E2 -1751.766} C_VEL
LIN {X 0,Y 580.266,Z 116.199,A -85,B 0,C 180,E1 -1754.626,E2 -1754.626} C_VEL
LIN {X 0,Y 580.283,Z 116.204,A -85,B 0,C 180,E1 -1757.628,E2 -1757.628} C_VEL
LIN {X 0,Y 580.291,Z 116.2,A -85,B 0,C 180,E1 -1760.067,E2 -1760.067} C_VEL
LIN {X 0,Y 580.296,Z 116.197,A -85,B 0,C 180,E1 -1763.066,E2 -1763.066} C_VEL
LIN {X 0,Y 580.313,Z 116.195,A -85,B 0,C 180,E1 -1766.145,E2 -1766.145} C_VEL
LIN {X 0,Y 580.285,Z 116.196,A -85,B 0,C 180,E1 -1768.615,E2 -1768.615} C_VEL
LIN {X 0,Y 580.29,Z 116.199,A -85,B 0,C 180,E1 -1771.024,E2 -1771.024} C_VEL
LIN {X 0,Y 580.289,Z 116.202,A -85,B 0,C 180,E1 -1773.666,E2 -1773.666} C_VEL
LIN {X 0,Y 580.297,Z 116.2,A -85,B 0,C 180,E1 -1775.684,E2 -1775.684} C_VEL
LIN {X 0,Y 580.272,Z 116.2,A -85,B 0,C 180,E1 -1777.948,E2 -1777.948} C_VEL
LIN {X 0,Y 580.317,Z 116.197,A -85,B 0,C 180,E1 -1780.914,E2 -1780.914} C_VEL
LIN {X 0,Y 580.274,Z 116.199,A -85,B 0,C 180,E1 -1783.826,E2 -1783.826} C_VEL
LIN {X 0,Y 580.324,Z 116.192,A -85,B 0,C 180,E1 -1785.983,E2 -1785.983} C_VEL
LIN {X 0,Y 580.303,Z 116.2,A -85,B 0,C 180,E1 -1788.827,E2 -1788.827} C_VEL
LIN {X 0,Y 580.326,Z 116.193,A -85,B 0,C 180,E1 -1791.644,E2 -1791.644} C_VEL
LIN {X 0,Y 580.329,Z 116.193,A -85,B 0,C 180,E1 -1794.441,E2 -1794.441} C_VEL
LIN {X 0,Y 580.334,Z 116.196,A -85,B 0,C 180,E1 -1797.224,E2 -1797.224} C_VEL
LIN {X 0,Y 580.352,Z 116.188,A -85,B 0,C 180,E1 -1800,E2 -1800} C_VEL
LIN {X 0,Y 580.337,Z 116.2,A -85,B 0,C 180,E1 -1802.777,E2 -1802.777} C_VEL
LIN {X 0,Y 580.326,Z 116.192,A -85,B 0,C 180,E1 -1805.56,E2 -1805.56} C_VEL
LIN {X 0,Y 580.333,Z 116.195,A -85,B 0,C 180,E1 -1808.356,E2 -1808.356} C_VEL
LIN {X 0,Y 580.299,Z 116.197,A -85,B 0,C 180,E1 -1811.191,E2 -1811.191} C_VEL
LIN {X 0,Y 580.324,Z 116.194,A -85,B 0,C 180,E1 -1814.017,E2 -1814.017} C_VEL
LIN {X 0,Y 580.311,Z 116.197,A -85,B 0,C 180,E1 -1816.914,E2 -1816.914} C_VEL
LIN {X 0,Y 580.304,Z 116.196,A -85,B 0,C 180,E1 -1819.823,E2 -1819.823} C_VEL
LIN {X 0,Y 580.29,Z 116.199,A -85,B 0,C 180,E1 -1822.803,E2 -1822.803} C_VEL
LIN {X 0,Y 580.306,Z 116.194,A -85,B 0,C 180,E1 -1825.08,E2 -1825.08} C_VEL
LIN {X 0,Y 580.298,Z 116.204,A -85,B 0,C 180,E1 -1828.186,E2 -1828.186} C_VEL
LIN {X 0,Y 580.284,Z 116.199,A -85,B 0,C 180,E1 -1830.695,E2 -1830.695} C_VEL
LIN {X 0,Y 580.303,Z 116.194,A -85,B 0,C 180,E1 -1833.317,E2 -1833.317} C_VEL
LIN {X 0,Y 580.245,Z 116.206,A -85,B 0,C 180,E1 -1835.757,E2 -1835.757} C_VEL
LIN {X 0,Y 580.289,Z 116.204,A -85,B 0,C 180,E1 -1838.147,E2 -1838.147} C_VEL
LIN {X 0,Y 580.3,Z 116.195,A -85,B 0,C 180,E1 -1840.844,E2 -1840.844} C_VEL
LIN {X 0,Y 580.28,Z 116.203,A -85,B 0,C 180,E1 -1843.658,E2 -1843.658} C_VEL
LIN {X 0,Y 580.278,Z 116.198,A -85,B 0,C 180,E1 -1846.61,E2 -1846.61} C_VEL
LIN {X 0,Y 580.3,Z 116.196,A -85,B 0,C 180,E1 -1849.157,E2 -1849.157} C_VEL
LIN {X 0,Y 580.292,Z 116.203,A -85,B 0,C 180,E1 -1851.927,E2 -1851.927} C_VEL
LIN {X 0,Y 580.251,Z 116.201,A -85,B 0,C 180,E1 -1854.453,E2 -1854.453} C_VEL
LIN {X 0,Y 580.292,Z 116.197,A -85,B 0,C 180,E1 -1856.976,E2 -1856.976} C_VEL
LIN {X 0,Y 580.296,Z 116.203,A -85,B 0,C 180,E1 -1859.425,E2 -1859.425} C_VEL
LIN {X 0,Y 580.3,Z 116.197,A -85,B 0,C 180,E1 -1862.142,E2 -1862.142} C_VEL
LIN {X 0,Y 580.323,Z 116.201,A -85,B 0,C 180,E1 -1865.27,E2 -1865.27} C_VEL
LIN {X 0,Y 580.35,Z 116.378,A -85,B 0,C 180,E1 -1865.924,E2 -1865.924} C_VEL
LIN {X 0,Y 580.982,Z 120.239,A -85,B 0,C 180,E1 -1866.473,E2 -1866.473} C_VEL
LIN {X 0,Y 580.847,Z 139.724,A -85,B 0,C 180,E1 -1869.088,E2 -1869.088} C_VEL
LIN {X 0,Y 580.705,Z 161.688,A -85,B 0,C 180,E1 -1872.025,E2 -1872.025} C_VEL
LIN {X 0,Y 580.484,Z 182.159,A -85,B 0,C 180,E1 -1874.733,E2 -1874.733} C_VEL
LIN {X 0,Y 580.401,Z 194.357,A -85,B 0,C 180,E1 -1876.331,E2 -1876.331} C_VEL
LIN {X 0,Y 580.963,Z 200.531,A -85,B 0,C 180,E1 -1876.423,E2 -1876.423} C_VEL
LIN {X 0,Y 580.809,Z 302.961,A -85,B 0,C 180,E1 -1877.708,E2 -1877.708} C_VEL
LIN {X 0,Y 580.726,Z 316.228,A -85,B 0,C 180,E1 -1878.017,E2 -1878.017} C_VEL
LIN {X 0,Y 580.656,Z 328.382,A -85,B 0,C 180,E1 -1878.436,E2 -1878.436} C_VEL
LIN {X 0,Y 580.579,Z 340.632,A -85,B 0,C 180,E1 -1879.009,E2 -1879.009} C_VEL
LIN {X 0,Y 580.441,Z 352.205,A -85,B 0,C 180,E1 -1879.712,E2 -1879.712} C_VEL
LIN {X 0,Y 580.345,Z 362.604,A -85,B 0,C 180,E1 -1880.503,E2 -1880.503} C_VEL
LIN {X 0,Y 580.271,Z 371.115,A -85,B 0,C 180,E1 -1881.293,E2 -1881.293} C_VEL
LIN {X 0,Y 580.222,Z 378.963,A -85,B 0,C 180,E1 -1882.168,E2 -1882.168} C_VEL
LIN {X 0,Y 580.153,Z 386.653,A -85,B 0,C 180,E1 -1883.222,E2 -1883.222} C_VEL
LIN {X 0,Y 580.139,Z 393.681,A -85,B 0,C 180,E1 -1884.439,E2 -1884.439} C_VEL
LIN {X 0,Y 580.108,Z 398.373,A -85,B 0,C 180,E1 -1885.484,E2 -1885.484} C_VEL
LIN {X 0,Y 580.123,Z 401.958,A -85,B 0,C 180,E1 -1886.528,E2 -1886.528} C_VEL
LIN {X 0,Y 580.043,Z 403.809,A -85,B 0,C 180,E1 -1887.222,E2 -1887.222} C_VEL
LIN {X 0,Y 580.04,Z 405.198,A -85,B 0,C 180,E1 -1887.917,E2 -1887.917} C_VEL
LIN {X 0,Y 580.04,Z 406.785,A -85,B 0,C 180,E1 -1889.306,E2 -1889.306} C_VEL
LIN {X 0,Y 580.037,Z 407,A -85,B 0,C 180,E1 -1890,E2 -1890} C_VEL
LIN {X 0,Y 580.047,Z 406.186,A -85,B 0,C 180,E1 -1891.389,E2 -1891.389} C_VEL
LIN {X 0,Y 580.04,Z 405.199,A -85,B 0,C 180,E1 -1892.083,E2 -1892.083} C_VEL
LIN {X 0,Y 580.043,Z 403.809,A -85,B 0,C 180,E1 -1892.778,E2 -1892.778} C_VEL
LIN {X 0,Y 580.11,Z 400.895,A -85,B 0,C 180,E1 -1893.821,E2 -1893.821} C_VEL
LIN {X 0,Y 580.053,Z 396.948,A -85,B 0,C 180,E1 -1894.866,E2 -1894.866} C_VEL
LIN {X 0,Y 580.139,Z 390.875,A -85,B 0,C 180,E1 -1896.085,E2 -1896.085} C_VEL
LIN {X 0,Y 580.184,Z 384.236,A -85,B 0,C 180,E1 -1897.133,E2 -1897.133} C_VEL
LIN {X 0,Y 580.25,Z 375.989,A -85,B 0,C 180,E1 -1898.182,E2 -1898.182} C_VEL
LIN {X 0,Y 580.308,Z 367.536,A -85,B 0,C 180,E1 -1899.059,E2 -1899.059} C_VEL
LIN {X 0,Y 580.422,Z 357.095,A -85,B 0,C 180,E1 -1899.936,E2 -1899.936} C_VEL
LIN {X 0,Y 580.506,Z 346.75,A -85,B 0,C 180,E1 -1900.64,E2 -1900.64} C_VEL
LIN {X 0,Y 580.597,Z 335.243,A -85,B 0,C 180,E1 -1901.264,E2 -1901.264} C_VEL
LIN {X 0,Y 580.683,Z 322.464,A -85,B 0,C 180,E1 -1901.785,E2 -1901.785} C_VEL
LIN {X 0,Y 580.777,Z 309.423,A -85,B 0,C 180,E1 -1902.16,E2 -1902.16} C_VEL
LIN {X 0,Y 580.84,Z 297.066,A -85,B 0,C 180,E1 -1902.38,E2 -1902.38} C_VEL
LIN {X 0,Y 580.802,Z 197.136,A -85,B 0,C 180,E1 -1903.623,E2 -1903.623} C_VEL
LIN {X 0,Y 580.407,Z 194.268,A -85,B 0,C 180,E1 -1903.68,E2 -1903.68} C_VEL
LIN {X 0,Y 580.602,Z 171.237,A -85,B 0,C 180,E1 -1906.708,E2 -1906.708} C_VEL
LIN {X 0,Y 580.731,Z 152.004,A -85,B 0,C 180,E1 -1909.273,E2 -1909.273} C_VEL
LIN {X 0,Y 580.87,Z 132.576,A -85,B 0,C 180,E1 -1911.842,E2 -1911.842} C_VEL
LIN {X 0,Y 580.928,Z 119.811,A -85,B 0,C 180,E1 -1913.53,E2 -1913.53} C_VEL
LIN {X 0,Y 580.34,Z 116.198,A -85,B 0,C 180,E1 -1914.03,E2 -1914.03} C_VEL
LIN {X 0,Y 580.28,Z 116.206,A -85,B 0,C 180,E1 -1916.623,E2 -1916.623} C_VEL
LIN {X 0,Y 580.305,Z 116.196,A -85,B 0,C 180,E1 -1919.31,E2 -1919.31} C_VEL
LIN {X 0,Y 580.302,Z 116.205,A -85,B 0,C 180,E1 -1922.201,E2 -1922.201} C_VEL
LIN {X 0,Y 580.291,Z 116.199,A -85,B 0,C 180,E1 -1924.696,E2 -1924.696} C_VEL
LIN {X 0,Y 580.303,Z 116.195,A -85,B 0,C 180,E1 -1927.268,E2 -1927.268} C_VEL
LIN {X 0,Y 580.295,Z 116.202,A -85,B 0,C 180,E1 -1930.27,E2 -1930.27} C_VEL
LIN {X 0,Y 580.28,Z 116.198,A -85,B 0,C 180,E1 -1932.706,E2 -1932.706} C_VEL
LIN {X 0,Y 580.274,Z 116.204,A -85,B 0,C 180,E1 -1935.609,E2 -1935.609} C_VEL
LIN {X 0,Y 580.293,Z 116.198,A -85,B 0,C 180,E1 -1938.232,E2 -1938.232} C_VEL
LIN {X 0,Y 580.281,Z 116.197,A -85,B 0,C 180,E1 -1940.965,E2 -1940.965} C_VEL
LIN {X 0,Y 580.271,Z 116.207,A -85,B 0,C 180,E1 -1943.596,E2 -1943.596} C_VEL
LIN {X 0,Y 580.285,Z 116.198,A -85,B 0,C 180,E1 -1946.143,E2 -1946.143} C_VEL
LIN {X 0,Y 580.276,Z 116.197,A -85,B 0,C 180,E1 -1948.614,E2 -1948.614} C_VEL
LIN {X 0,Y 580.294,Z 116.2,A -85,B 0,C 180,E1 -1951.024,E2 -1951.024} C_VEL
LIN {X 0,Y 580.292,Z 116.2,A -85,B 0,C 180,E1 -1953.666,E2 -1953.666} C_VEL
LIN {X 0,Y 580.294,Z 116.199,A -85,B 0,C 180,E1 -1955.683,E2 -1955.683} C_VEL
LIN {X 0,Y 580.27,Z 116.199,A -85,B 0,C 180,E1 -1957.947,E2 -1957.947} C_VEL
LIN {X 0,Y 580.298,Z 116.202,A -85,B 0,C 180,E1 -1960.913,E2 -1960.913} C_VEL
LIN {X 0,Y 580.265,Z 116.199,A -85,B 0,C 180,E1 -1963.825,E2 -1963.825} C_VEL
LIN {X 0,Y 580.268,Z 116.206,A -85,B 0,C 180,E1 -1966.696,E2 -1966.696} C_VEL
LIN {X 0,Y 580.309,Z 116.203,A -85,B 0,C 180,E1 -1968.827,E2 -1968.827} C_VEL
LIN {X 0,Y 580.309,Z 116.194,A -85,B 0,C 180,E1 -1971.643,E2 -1971.643} C_VEL
LIN {X 0,Y 580.331,Z 116.198,A -85,B 0,C 180,E1 -1974.44,E2 -1974.44} C_VEL
LIN {X 0,Y 580.342,Z 116.192,A -85,B 0,C 180,E1 -1977.918,E2 -1977.918} C_VEL
LIN {X 0,Y 580.356,Z 116.195,A -85,B 0,C 180,E1 -1980.694,E2 -1980.694} C_VEL
LIN {X 0,Y 580.326,Z 116.197,A -85,B 0,C 180,E1 -1982.776,E2 -1982.776} C_VEL
LIN {X 0,Y 580.314,Z 116.195,A -85,B 0,C 180,E1 -1985.56,E2 -1985.56} C_VEL
LIN {X 0,Y 580.317,Z 116.344,A -85,B 0,C 180,E1 -1987.48,E2 -1987.48} C_VEL
LIN {X 0,Y 580.281,Z 130.096,A -85,B 0,C 180,E1 -1990.114,E2 -1990.114} C_VEL
LIN {X 0,Y 580.299,Z 136.836,A -85,B 0,C 180,E1 -1991.394,E2 -1991.394} C_VEL
LIN {X 0,Y 580.969,Z 142.717,A -85,B 0,C 180,E1 -1991.495,E2 -1991.495} C_VEL
LIN {X 0,Y 580.833,Z 221.154,A -85,B 0,C 180,E1 -1992.467,E2 -1992.467} C_VEL
LIN {X 0,Y 580.168,Z 227.015,A -85,B 0,C 180,E1 -1992.521,E2 -1992.521} C_VEL
LIN {X 0,Y 574.668,Z 245.011,A -85,B 0,C 180,E1 -1992.651,E2 -1992.651} C_VEL
LIN {X 0,Y 573.888,Z 249.776,A -85,B 0,C 180,E1 -1992.741,E2 -1992.741} C_VEL
LIN {X 0,Y 573.817,Z 251.677,A -85,B 0,C 180,E1 -1992.79,E2 -1992.79} C_VEL
LIN {X 0,Y 573.713,Z 264.372,A -85,B 0,C 180,E1 -1993.188,E2 -1993.188} C_VEL
LIN {X 0,Y 573.632,Z 273.187,A -85,B 0,C 180,E1 -1993.551,E2 -1993.551} C_VEL
LIN {X 0,Y 573.491,Z 283.711,A -85,B 0,C 180,E1 -1994.097,E2 -1994.097} C_VEL
LIN {X 0,Y 573.418,Z 292.253,A -85,B 0,C 180,E1 -1994.639,E2 -1994.639} C_VEL
LIN {X 0,Y 573.345,Z 300.731,A -85,B 0,C 180,E1 -1995.28,E2 -1995.28} C_VEL
LIN {X 0,Y 573.26,Z 308.868,A -85,B 0,C 180,E1 -1996.012,E2 -1996.012} C_VEL
LIN {X 0,Y 573.174,Z 316.958,A -85,B 0,C 180,E1 -1996.883,E2 -1996.883} C_VEL
LIN {X 0,Y 573.121,Z 324.411,A -85,B 0,C 180,E1 -1997.852,E2 -1997.852} C_VEL
LIN {X 0,Y 573.072,Z 330.98,A -85,B 0,C 180,E1 -1998.902,E2 -1998.902} C_VEL
LIN {X 0,Y 573.029,Z 336.784,A -85,B 0,C 180,E1 -2000.084,E2 -2000.084} C_VEL
LIN {X 0,Y 572.987,Z 340.993,A -85,B 0,C 180,E1 -2001.222,E2 -2001.222} C_VEL
LIN {X 0,Y 572.95,Z 344.015,A -85,B 0,C 180,E1 -2002.349,E2 -2002.349} C_VEL
LIN {X 0,Y 572.934,Z 345.487,A -85,B 0,C 180,E1 -2003.112,E2 -2003.112} C_VEL
LIN {X 0,Y 572.926,Z 346.442,A -85,B 0,C 180,E1 -2003.879,E2 -2003.879} C_VEL
LIN {X 0,Y 572.929,Z 346.952,A -85,B 0,C 180,E1 -2004.804,E2 -2004.804} C_VEL
LIN {X 0,Y 572.945,Z 346.449,A -85,B 0,C 180,E1 -2006.205,E2 -2006.205} C_VEL
LIN {X 0,Y 572.94,Z 345.464,A -85,B 0,C 180,E1 -2006.991,E2 -2006.991} C_VEL
LIN {X 0,Y 572.957,Z 343.52,A -85,B 0,C 180,E1 -2007.973,E2 -2007.973} C_VEL
LIN {X 0,Y 573.025,Z 339.266,A -85,B 0,C 180,E1 -2009.379,E2 -2009.379} C_VEL
LIN {X 0,Y 573.029,Z 334.404,A -85,B 0,C 180,E1 -2010.52,E2 -2010.52} C_VEL
LIN {X 0,Y 573.09,Z 328.422,A -85,B 0,C 180,E1 -2011.618,E2 -2011.618} C_VEL
LIN {X 0,Y 573.123,Z 321.424,A -85,B 0,C 180,E1 -2012.653,E2 -2012.653} C_VEL
LIN {X 0,Y 573.237,Z 312.894,A -85,B 0,C 180,E1 -2013.673,E2 -2013.673} C_VEL
LIN {X 0,Y 573.326,Z 304.538,A -85,B 0,C 180,E1 -2014.49,E2 -2014.49} C_VEL
LIN {X 0,Y 573.414,Z 294.67,A -85,B 0,C 180,E1 -2015.28,E2 -2015.28} C_VEL
LIN {X 0,Y 573.506,Z 285.492,A -85,B 0,C 180,E1 -2015.888,E2 -2015.888} C_VEL
LIN {X 0,Y 573.61,Z 274.888,A -85,B 0,C 180,E1 -2016.458,E2 -2016.458} C_VEL
LIN {X 0,Y 573.707,Z 264.741,A -85,B 0,C 180,E1 -2016.888,E2 -2016.888} C_VEL
LIN {X 0,Y 573.787,Z 253.953,A -85,B 0,C 180,E1 -2017.236,E2 -2017.236} C_VEL
LIN {X 0,Y 573.835,Z 241.679,A -85,B 0,C 180,E1 -2017.508,E2 -2017.508} C_VEL
LIN {X 0,Y 573.896,Z 141.058,A -85,B 0,C 180,E1 -2018.786,E2 -2018.786} C_VEL
LIN {X 0,Y 573.226,Z 136.857,A -85,B 0,C 180,E1 -2018.864,E2 -2018.864} C_VEL
LIN {X 0,Y 573.346,Z 122.646,A -85,B 0,C 180,E1 -2021.606,E2 -2021.606} C_VEL
LIN {X 0,Y 573.273,Z 117.074,A -85,B 0,C 180,E1 -2022.732,E2 -2022.732} C_VEL
LIN {X 0,Y 573.236,Z 117.084,A -85,B 0,C 180,E1 -2025.666,E2 -2025.666} C_VEL
LIN {X 0,Y 573.239,Z 117.074,A -85,B 0,C 180,E1 -2028.543,E2 -2028.543} C_VEL
LIN {X 0,Y 573.242,Z 117.078,A -85,B 0,C 180,E1 -2031.298,E2 -2031.298} C_VEL
LIN {X 0,Y 573.212,Z 117.081,A -85,B 0,C 180,E1 -2034.018,E2 -2034.018} C_VEL
LIN {X 0,Y 573.238,Z 117.074,A -85,B 0,C 180,E1 -2036.516,E2 -2036.516} C_VEL
LIN {X 0,Y 573.224,Z 117.08,A -85,B 0,C 180,E1 -2039.118,E2 -2039.118} C_VEL
LIN {X 0,Y 573.251,Z 117.075,A -85,B 0,C 180,E1 -2041.971,E2 -2041.971} C_VEL
LIN {X 0,Y 573.252,Z 117.073,A -85,B 0,C 180,E1 -2044.59,E2 -2044.59} C_VEL
LIN {X 0,Y 573.236,Z 117.079,A -85,B 0,C 180,E1 -2047.662,E2 -2047.662} C_VEL
LIN {X 0,Y 573.265,Z 117.073,A -85,B 0,C 180,E1 -2050.67,E2 -2050.67} C_VEL
LIN {X 0,Y 573.246,Z 117.076,A -85,B 0,C 180,E1 -2053.621,E2 -2053.621} C_VEL
LIN {X 0,Y 573.273,Z 117.071,A -85,B 0,C 180,E1 -2055.807,E2 -2055.807} C_VEL
LIN {X 0,Y 573.262,Z 117.076,A -85,B 0,C 180,E1 -2058.745,E2 -2058.745} C_VEL
LIN {X 0,Y 573.282,Z 117.071,A -85,B 0,C 180,E1 -2061.54,E2 -2061.54} C_VEL
LIN {X 0,Y 573.297,Z 117.069,A -85,B 0,C 180,E1 -2064.372,E2 -2064.372} C_VEL
LIN {X 0,Y 573.314,Z 117.065,A -85,B 0,C 180,E1 -2067.892,E2 -2067.892} C_VEL
LIN {X 0,Y 573.335,Z 117.071,A -85,B 0,C 180,E1 -2070.702,E2 -2070.702} C_VEL
LIN {X 0,Y 573.305,Z 117.075,A -85,B 0,C 180,E1 -2072.81,E2 -2072.81} C_VEL
LIN {X 0,Y 573.293,Z 117.067,A -85,B 0,C 180,E1 -2075.628,E2 -2075.628} C_VEL
LIN {X 0,Y 573.289,Z 117.075,A -85,B 0,C 180,E1 -2078.459,E2 -2078.459} C_VEL
LIN {X 0,Y 573.27,Z 117.071,A -85,B 0,C 180,E1 -2081.312,E2 -2081.312} C_VEL
LIN {X 0,Y 573.28,Z 117.078,A -85,B 0,C 180,E1 -2084.424,E2 -2084.424} C_VEL
LIN {X 0,Y 573.256,Z 117.073,A -85,B 0,C 180,E1 -2087.111,E2 -2087.111} C_VEL
LIN {X 0,Y 573.25,Z 117.078,A -85,B 0,C 180,E1 -2090.076,E2 -2090.076} C_VEL
LIN {X 0,Y 573.232,Z 117.075,A -85,B 0,C 180,E1 -2093.099,E2 -2093.099} C_VEL
LIN {X 0,Y 573.253,Z 117.073,A -85,B 0,C 180,E1 -2095.41,E2 -2095.41} C_VEL
LIN {X 0,Y 573.248,Z 117.08,A -85,B 0,C 180,E1 -2098.029,E2 -2098.029} C_VEL
LIN {X 0,Y 573.241,Z 117.075,A -85,B 0,C 180,E1 -2100.885,E2 -2100.885} C_VEL
LIN {X 0,Y 573.259,Z 117.074,A -85,B 0,C 180,E1 -2103.524,E2 -2103.524} C_VEL
LIN {X 0,Y 573.254,Z 117.082,A -85,B 0,C 180,E1 -2106.048,E2 -2106.048} C_VEL
LIN {X 0,Y 573.247,Z 117.074,A -85,B 0,C 180,E1 -2108.701,E2 -2108.701} C_VEL
LIN {X 0,Y 573.251,Z 117.077,A -85,B 0,C 180,E1 -2111.596,E2 -2111.596} C_VEL
LIN {X 0,Y 573.237,Z 117.077,A -85,B 0,C 180,E1 -2114.333,E2 -2114.333} C_VEL
LIN {X 0,Y 573.238,Z 117.078,A -85,B 0,C 180,E1 -2117.358,E2 -2117.358} C_VEL
LIN {X 0,Y 573.245,Z 117.075,A -85,B 0,C 180,E1 -2120.393,E2 -2120.393} C_VEL
LIN {X 0,Y 573.25,Z 117.075,A -85,B 0,C 180,E1 -2123.078,E2 -2123.078} C_VEL
LIN {X 0,Y 573.265,Z 117.08,A -85,B 0,C 180,E1 -2125.671,E2 -2125.671} C_VEL
LIN {X 0,Y 573.247,Z 117.075,A -85,B 0,C 180,E1 -2128.185,E2 -2128.185} C_VEL
LIN {X 0,Y 573.261,Z 117.072,A -85,B 0,C 180,E1 -2130.634,E2 -2130.634} C_VEL
LIN {X 0,Y 573.249,Z 117.076,A -85,B 0,C 180,E1 -2133.024,E2 -2133.024} C_VEL
LIN {X 0,Y 573.272,Z 117.08,A -85,B 0,C 180,E1 -2135.366,E2 -2135.366} C_VEL
LIN {X 0,Y 573.227,Z 117.076,A -85,B 0,C 180,E1 -2138.42,E2 -2138.42} C_VEL
LIN {X 0,Y 573.276,Z 117.072,A -85,B 0,C 180,E1 -2140.728,E2 -2140.728} C_VEL
LIN {X 0,Y 573.247,Z 117.077,A -85,B 0,C 180,E1 -2143.622,E2 -2143.622} C_VEL
LIN {X 0,Y 573.271,Z 117.072,A -85,B 0,C 180,E1 -2145.807,E2 -2145.807} C_VEL
LIN {X 0,Y 573.261,Z 117.076,A -85,B 0,C 180,E1 -2148.745,E2 -2148.745} C_VEL
LIN {X 0,Y 573.282,Z 117.072,A -85,B 0,C 180,E1 -2151.541,E2 -2151.541} C_VEL
LIN {X 0,Y 573.297,Z 117.068,A -85,B 0,C 180,E1 -2154.372,E2 -2154.372} C_VEL
LIN {X 0,Y 573.314,Z 117.065,A -85,B 0,C 180,E1 -2157.893,E2 -2157.893} C_VEL
LIN {X 0,Y 573.333,Z 117.07,A -85,B 0,C 180,E1 -2160.703,E2 -2160.703} C_VEL
LIN {X 0,Y 573.303,Z 117.077,A -85,B 0,C 180,E1 -2162.811,E2 -2162.811} C_VEL
LIN {X 0,Y 573.294,Z 117.067,A -85,B 0,C 180,E1 -2165.628,E2 -2165.628} C_VEL
LIN {X 0,Y 573.289,Z 117.074,A -85,B 0,C 180,E1 -2168.46,E2 -2168.46} C_VEL
LIN {X 0,Y 573.271,Z 117.071,A -85,B 0,C 180,E1 -2171.312,E2 -2171.312} C_VEL
LIN {X 0,Y 573.272,Z 117.074,A -85,B 0,C 180,E1 -2174.193,E2 -2174.193} C_VEL
LIN {X 0,Y 573.257,Z 117.073,A -85,B 0,C 180,E1 -2177.112,E2 -2177.112} C_VEL
LIN {X 0,Y 573.252,Z 117.077,A -85,B 0,C 180,E1 -2180.077,E2 -2180.077} C_VEL
LIN {X 0,Y 573.234,Z 117.076,A -85,B 0,C 180,E1 -2183.1,E2 -2183.1} C_VEL
LIN {X 0,Y 573.254,Z 117.072,A -85,B 0,C 180,E1 -2185.41,E2 -2185.41} C_VEL
LIN {X 0,Y 573.25,Z 117.079,A -85,B 0,C 180,E1 -2188.029,E2 -2188.029} C_VEL
LIN {X 0,Y 573.246,Z 117.083,A -85,B 0,C 180,E1 -2190.176,E2 -2190.176} C_VEL
LIN {X 0,Y 573.253,Z 117.075,A -85,B 0,C 180,E1 -2192.645,E2 -2192.645} C_VEL
LIN {X 0,Y 573.206,Z 117.078,A -85,B 0,C 180,E1 -2195.188,E2 -2195.188} C_VEL
LIN {X 0,Y 573.236,Z 117.08,A -85,B 0,C 180,E1 -2197.808,E2 -2197.808} C_VEL
LIN {X 0,Y 573.27,Z 117.073,A -85,B 0,C 180,E1 -2200.529,E2 -2200.529} C_VEL
LIN {X 0,Y 573.245,Z 117.079,A -85,B 0,C 180,E1 -2203.669,E2 -2203.669} C_VEL
LIN {X 0,Y 573.24,Z 117.075,A -85,B 0,C 180,E1 -2206.641,E2 -2206.641} C_VEL
LIN {X 0,Y 573.26,Z 117.076,A -85,B 0,C 180,E1 -2209.477,E2 -2209.477} C_VEL
LIN {X 0,Y 573.237,Z 117.078,A -85,B 0,C 180,E1 -2212.193,E2 -2212.193} C_VEL
LIN {X 0,Y 573.236,Z 117.078,A -85,B 0,C 180,E1 -2215.229,E2 -2215.229} C_VEL
LIN {X 0,Y 573.253,Z 117.08,A -85,B 0,C 180,E1 -2217.772,E2 -2217.772} C_VEL
LIN {X 0,Y 573.265,Z 117.071,A -85,B 0,C 180,E1 -2220.635,E2 -2220.635} C_VEL
LIN {X 0,Y 573.252,Z 117.076,A -85,B 0,C 180,E1 -2223.024,E2 -2223.024} C_VEL
LIN {X 0,Y 573.285,Z 117.128,A -85,B 0,C 180,E1 -2225.753,E2 -2225.753} C_VEL
LIN {X 0,Y 574.08,Z 122.143,A -85,B 0,C 180,E1 -2226.473,E2 -2226.473} C_VEL
LIN {X 0,Y 573.867,Z 142.219,A -85,B 0,C 180,E1 -2229.197,E2 -2229.197} C_VEL
LIN {X 0,Y 573.711,Z 164.417,A -85,B 0,C 180,E1 -2232.167,E2 -2232.167} C_VEL
LIN {X 0,Y 573.475,Z 184.889,A -85,B 0,C 180,E1 -2234.905,E2 -2234.905} C_VEL
LIN {X 0,Y 573.41,Z 194.357,A -85,B 0,C 180,E1 -2236.161,E2 -2236.161} C_VEL
LIN {X 0,Y 574.056,Z 200.531,A -85,B 0,C 180,E1 -2236.256,E2 -2236.256} C_VEL
LIN {X 0,Y 573.886,Z 302.961,A -85,B 0,C 180,E1 -2237.558,E2 -2237.558} C_VEL
LIN {X 0,Y 573.778,Z 316.228,A -85,B 0,C 180,E1 -2237.87,E2 -2237.87} C_VEL
LIN {X 0,Y 573.682,Z 329.503,A -85,B 0,C 180,E1 -2238.339,E2 -2238.339} C_VEL
LIN {X 0,Y 573.586,Z 340.641,A -85,B 0,C 180,E1 -2238.874,E2 -2238.874} C_VEL
LIN {X 0,Y 573.428,Z 352.202,A -85,B 0,C 180,E1 -2239.585,E2 -2239.585} C_VEL
LIN {X 0,Y 573.332,Z 362.606,A -85,B 0,C 180,E1 -2240.386,E2 -2240.386} C_VEL
LIN {X 0,Y 573.241,Z 371.116,A -85,B 0,C 180,E1 -2241.185,E2 -2241.185} C_VEL
LIN {X 0,Y 573.161,Z 378.963,A -85,B 0,C 180,E1 -2242.071,E2 -2242.071} C_VEL
LIN {X 0,Y 573.072,Z 386.957,A -85,B 0,C 180,E1 -2243.186,E2 -2243.186} C_VEL
LIN {X 0,Y 573.07,Z 393.681,A -85,B 0,C 180,E1 -2244.37,E2 -2244.37} C_VEL
LIN {X 0,Y 573.028,Z 398.373,A -85,B 0,C 180,E1 -2245.428,E2 -2245.428} C_VEL
LIN {X 0,Y 573.022,Z 401.958,A -85,B 0,C 180,E1 -2246.484,E2 -2246.484} C_VEL
LIN {X 0,Y 572.959,Z 403.808,A -85,B 0,C 180,E1 -2247.188,E2 -2247.188} C_VEL
LIN {X 0,Y 572.946,Z 406.185,A -85,B 0,C 180,E1 -2248.594,E2 -2248.594} C_VEL
LIN {X 0,Y 572.938,Z 407,A -85,B 0,C 180,E1 -2250,E2 -2250} C_VEL
LIN {X 0,Y 572.946,Z 406.185,A -85,B 0,C 180,E1 -2251.406,E2 -2251.406} C_VEL
LIN {X 0,Y 572.94,Z 405.198,A -85,B 0,C 180,E1 -2252.109,E2 -2252.109} C_VEL
LIN {X 0,Y 572.959,Z 403.809,A -85,B 0,C 180,E1 -2252.813,E2 -2252.813} C_VEL
LIN {X 0,Y 573.015,Z 400.895,A -85,B 0,C 180,E1 -2253.868,E2 -2253.868} C_VEL
LIN {X 0,Y 572.963,Z 396.948,A -85,B 0,C 180,E1 -2254.926,E2 -2254.926} C_VEL
LIN {X 0,Y 573.065,Z 390.875,A -85,B 0,C 180,E1 -2256.16,E2 -2256.16} C_VEL
LIN {X 0,Y 573.12,Z 384.235,A -85,B 0,C 180,E1 -2257.221,E2 -2257.221} C_VEL
LIN {X 0,Y 573.201,Z 375.989,A -85,B 0,C 180,E1 -2258.283,E2 -2258.283} C_VEL
LIN {X 0,Y 573.287,Z 367.536,A -85,B 0,C 180,E1 -2259.171,E2 -2259.171} C_VEL
LIN {X 0,Y 573.427,Z 357.092,A -85,B 0,C 180,E1 -2260.059,E2 -2260.059} C_VEL
LIN {X 0,Y 573.544,Z 345.428,A -85,B 0,C 180,E1 -2260.853,E2 -2260.853} C_VEL
LIN {X 0,Y 573.652,Z 334.304,A -85,B 0,C 180,E1 -2261.446,E2 -2261.446} C_VEL
LIN {X 0,Y 573.746,Z 321.162,A -85,B 0,C 180,E1 -2261.974,E2 -2261.974} C_VEL
LIN {X 0,Y 573.874,Z 308.507,A -85,B 0,C 180,E1 -2262.331,E2 -2262.331} C_VEL
LIN {X 0,Y 573.94,Z 295.29,A -85,B 0,C 180,E1 -2262.554,E2 -2262.554} C_VEL
LIN {X 0,Y 573.916,Z 197.93,A -85,B 0,C 180,E1 -2263.78,E2 -2263.78} C_VEL
LIN {X 0,Y 573.414,Z 194.268,A -85,B 0,C 180,E1 -2263.85,E2 -2263.85} C_VEL
LIN {X 0,Y 573.604,Z 172.625,A -85,B 0,C 180,E1 -2266.731,E2 -2266.731} C_VEL
LIN {X 0,Y 573.718,Z 156.017,A -85,B 0,C 180,E1 -2268.943,E2 -2268.943} C_VEL
LIN {X 0,Y 573.887,Z 136.292,A -85,B 0,C 180,E1 -2271.555,E2 -2271.555} C_VEL
LIN {X 0,Y 573.992,Z 121.511,A -85,B 0,C 180,E1 -2273.526,E2 -2273.526} C_VEL
LIN {X 0,Y 573.3,Z 117.075,A -85,B 0,C 180,E1 -2274.151,E2 -2274.151} C_VEL
LIN {X 0,Y 573.252,Z 117.077,A -85,B 0,C 180,E1 -2276.976,E2 -2276.976} C_VEL
LIN {X 0,Y 573.25,Z 117.076,A -85,B 0,C 180,E1 -2279.488,E2 -2279.488} C_VEL
LIN {X 0,Y 573.257,Z 117.077,A -85,B 0,C 180,E1 -2282.645,E2 -2282.645} C_VEL
LIN {X 0,Y 573.209,Z 117.079,A -85,B 0,C 180,E1 -2285.188,E2 -2285.188} C_VEL
LIN {X 0,Y 573.24,Z 117.08,A -85,B 0,C 180,E1 -2287.807,E2 -2287.807} C_VEL
LIN {X 0,Y 573.248,Z 117.076,A -85,B 0,C 180,E1 -2290.525,E2 -2290.525} C_VEL
LIN {X 0,Y 573.243,Z 117.076,A -85,B 0,C 180,E1 -2293.359,E2 -2293.359} C_VEL
LIN {X 0,Y 573.248,Z 117.076,A -85,B 0,C 180,E1 -2296.331,E2 -2296.331} C_VEL
